// SIMATIC STEP 7 (V5.x) project BAS_20HSL
// CPU: CPU 414-5 H PN/DP(1)
// CPU: CPU 414-5 H PN/DP
// CPU: CPU 414-5 H PN/DP
// CPU: CPU 412-5 H PN/DP
// CPU: CPU 414-5 H PN/DP(1)
// station: Hardware
// station: B_PLC(MAIN)
// station: P_ADR_BUS
// station: Hardware
// station: P_ADR_BUS
// station: A_PLC
// station: IBP_PLC
// station: Hardware
// station: P_ADR_BUS
// program: S7 Program(2)
// program: S7 Program(1)
// program: S7 Program(1)
// program: S7 Program(5)
// program: S7 Program(9)

SYMBOL_TABLE
"CONTROL_DAT"	DB 1	DB 1
"MODBUS_HPARAM_PN_2"	DB 2	DB 2
"License DB"	DB 3	DB 3
"CPULINDB"	DB 30	DB 30
"SYS_Date_Time_D"	DB 34	DB 34	// 系统日期和时间设置和读取数据区
"FB200_DB"	DB 200	FB 200
"FB201_DB"	DB 201	FB 201
"MAIN-READ-SLAVE"	DB 202	DB 202
"MAIN-WRITE-SLAVE"	DB 203	DB 203
"MAIN-READ-IBP"	DB 204	DB 204
"MAIN-WRITE-IBP"	DB 205	DB 205
"DETAIL_DIAG_DB_RACK0"	DB 458	FB 315	// DB FOR SFB13
"DETAIL_DIAG_DB_RACK1"	DB 459	FB 315	// DB FOR SFB12
"DP_ERROR_RACK0"	DB 460	DB 460
"DP_ERROR_RESET_DB"	DB 461	DB 461
"DP_ERROR_FB1501"	DB 462	FB 1501
"DB_FOR_FB300"	DB 463	FB 300
"DP_VAT"	DB 464	DB 464
"DP_ERROR_RACK1"	DB 465	DB 465
"DP_ERROR1_RESET"	DB 466	DB 466
"DP_ERROR1_FB1501"	DB 467	FB 1501
"FB523_DB"	DB 523	FB 523
"LED"	DB 525	DB 525
"IDB_MODBUS"	DB 915	FB 915
"JOBLIST_DB"	DB 919	FB 919
"JOB_RESET_DB"	DB 921	FB 921
"AP_BMPSB"	DB 2005	DB 2005
"EPS21"	DB 2015	DB 2015
"E411_08_C"	DB 2025	DB 2025
"AT_AYSB4_WRITE"	DB 2033	DB 2033
"AT_AYSB4_READ"	DB 2035	DB 2035
"AT_aysb1_2_WRITE"	DB 2043	DB 2043
"AT_AYSB1_2_READ"	DB 2045	DB 2045
"AP_PSB_C1_C2"	DB 2055	DB 2055
"AT_FSB_3_4_PSD2"	DB 2065	DB 2065
"AP_PSB_C"	DB 2075	DB 2075
"EPS11"	DB 2095	DB 2095
"E411_01_02_N"	DB 2105	DB 2105
"AP_FSB_WRITE"	DB 2113	DB 2113
"AP_FSB_READ"	DB 2115	DB 2115
"AT_QJSB_WRITE"	DB 2123	DB 2123
"AT_QJSB_READ"	DB 2125	DB 2125
"HF3_IMCC_Read_DB2291"	DB 2291	DB 2291	// IMCC系统读取数据
"HF3_IMCC_Write_DB2292"	DB 2292	DB 2292	// IMCC系统写数据
"HF3_EPS_HMI"	DB 2501	FB 2501	// EPS_ToHMI
"IMCC_LOCK"	DB 2555	DB 2555
"MAIN_ToHMI"	DB 6002	DB 6002	// 发送数据至HMI
"ISCS_CONTROL"	DB 6003	DB 6003
"SLAVE_TO_HMI"	DB 6004	DB 6004
"HF3_DP_Statu_ToHMI"	DB 6009	DB 6009
"HF3_PLC_Statu_ToHMI"	DB 6010	DB 6010
"给上位_状态"	DB 6030	DB 6030
"HF4_Sum_SCtrl"	DB 6040	DB 6040
"HF4_Mode_DB"	DB 7004	DB 7004	// B端模式控制命令
"Maste_To_Slave_Mod_DB"	DB 7005	DB 7005
"MODE_REFUSE"	DB 7006	DB 7006
"P_RCV"	FB 12	FB 12	// Receive Data from CP340
"P_SEND"	FB 13	FB 13	// Send Data to CP340
"pid"	FB 41	FB 41
"TSEND"	FB 63	FB 63	// Send Data
"TRCV"	FB 64	FB 64	// Receive Data
"TCON"	FB 65	FB 65	// Connect
"TDISCON"	FB 66	FB 66	// Disconnect
"P_RESET"	FB 177	FB 177	// Reset Job for CP340
"S7400H-COM-MAIN-SLAVE"	FB 200	FB 200
"S7400H-COM-MAIN-IBP"	FB 201	FB 201
"S7400H-COM-SLAVE-MAIN"	FB 202	FB 202
"READ_ERROR"	FB 300	FB 300
"DETAIL_DP_DIAG"	FB 315	FB 315
"H_STATUS"	FB 523	FB 523	// Status H-System
"TCP_COMM"	FB 913	FB 913	// TCP Kommunikation
"MOD_CLI"	FB 914	FB 914
"MB_PNHCL"	FB 915	FB 915
"Job_List"	FB 919	FB 919
"JOB_RESET"	FB 921	FB 921
"MODMAS_STEP7_CP340_L"	FB 1071	FB 1071
"com_check"	FB 1501	FB 1501
"HF3_PID_FB2005"	FB 2005	FB 2005	// PID处理功能块
"HF3_RunFaultSum"	FB 2006	FB 2006	// 运行时间故障次数统计
"HF3_EPS_FB2501"	FB 2501	FB 2501	// EPS主程序段
"HF3_EPS_FB2502"	FB 2502	FB 2502	// EPS功能块
"HF3_IMCC_CommOK_FB2512"	FB 2512	FB 2512	// IMCC心跳
"HF3_IMCC_CommOK_FB2513"	FB 2513	FB 2513
"HF3_LSQK_FB2521"	FB 2521	FB 2521	// 冷水群控程序段
"HF3_LSQK_FB2522"	FB 2522	FB 2522	// LSQK功能块
"HF3_JET_FB2531"	FB 2531	FB 2531	// 射流风机主程序端
"HF3_JET_FB2532"	FB 2532	FB 2532	// 射流风机功能块
"HF3_VRV_FB2541"	FB 2541	FB 2541	// 多联体空调主程序段
"HF3_VRV_FB2542"	FB 2542	FB 2542	// 多联体空调程序端
"HF3_SB_FB2551"	FB 2551	FB 2551	// 带控制水泵程序段
"HF3_SB_FB2552"	FB 2552	FB 2552	// 带控制水泵功能块
"HF3_3#SB_FB2561"	FB 2561	FB 2561	// 洞口水泵主程序段
"HF3_3#SB_FB2562"	FB 2562	FB 2562	// 洞口水泵功能块
"HF3_WSB_FB2581"	FB 2581	FB 2581	// 污水密闭提升
"HF3_WSB_FB2582"	FB 2582	FB 2582
"HF3_PSB_FB2591"	FB 2591	FB 2591	// 局部排水泵主程序
"HF3_PSB_FB2592"	FB 2592	FB 2592	// 排水泵DB转换
"HF3_UPS_FB2611"	FB 2611	FB 2611
"HF3_UPS_FB2612"	FB 2612	FB 2612
"HF3_DT_FB2621"	FB 2621	FB 2621	// 电梯
"HF3_DT_FB2622"	FB 2622	FB 2622	// 电梯
"HF3_FT_FB2631"	FB 2631	FB 2631	// 扶梯
"HF4_FT_FB2362"	FB 2632	FB 2632
"HF3_IMCC_TVF_FB2651"	FB 2651	FB 2651	// 隧道风机主程序段
"HF4_IMCC_TVF_FB2652"	FB 2652	FB 2652	// 隧道风机功能块
"HF3_IMCC_TEF_FB2661"	FB 2661	FB 2661	// 排热风机主程序
"HF3_IMCC_TEF_FB2662"	FB 2662	FB 2662	// 排热风机功能块
"HF3_IMCC_KT_FB2671"	FB 2671	FB 2671	// 大空调主程序
"HF3_IMCC_KT_FB2672"	FB 2672	FB 2672	// 空调机组功能块
"HF3_IMCC_HPF_FB2681"	FB 2681	FB 2681	// IMCC_HPF_主程序
"HF4_IMCC_HPF_FB2682"	FB 2682	FB 2682	// IMCC_HPF功能块
"HF3_IMCC_FJ_FB2691"	FB 2691	FB 2691	// 智能低压小风机
"HF3_IMCC_FJ_FB2692"	FB 2692	FB 2692	// 智能低压小风机功能块
"HF3_IMCC_DZ_FB2701"	FB 2701	FB 2701	// IMCC组合阀主程序
"HF3_IMCC_DZ_B2702"	FB 2702	FB 2702	// 电动组合风阀功能块
"HF3_IMCC_DT_FB2711"	FB 2711	FB 2711	// IMCC风量调节阀程序
"HF3_IMCC_DT_FB2712"	FB 2712	FB 2712	// IMCC风量调节阀块
"HF3_IMCC_D_FB2721"	FB 2721	FB 2721	// IMCC电动风阀主程序
"HF3_IMCC_D_FB2722"	FB 2722	FB 2722	// IMCC电动风阀功能块
"HF3_JH_YC_FB2731"	FB 2731	FB 2731	// 电子净化压差主程序
"HF3_DPH_FB2751"	FB 2751	FB 2751	// 二通阀主程序
"HF3_DPH_FB2752"	FB 2752	FB 2752	// 二通阀主程序
"HF3_FJ_FB2761"	FB 2761	FB 2761	// 高架站风机主程序段
"HF3_FJ_FB2762"	FB 2762	FB 2762	// 高架站风机
"HF3_FJPG_FB2771"	FB 2771	FB 2771	// 风机盘管主程序段
"HF3_FJPG_FB2772"	FB 2772	FB 2772	// 风机盘管功能块
"HF3_XFDF_FB2781"	FB 2781	FB 2781	// 手电一体蝶阀程序段
"HF2_XVDF_FB2782"	FB 2782	FB 2782	// 手电一体蝶阀功能块
"HF3_EPS_WLE_FB2791"	FB 2791	FB 2791	// 区间疏散指示
"HF3_EPS_WLE_FB2792"	FB 2792	FB 2792	// 区间疏散指示功能块
"HF3_D_FB2801"	FB 2801	FB 2801	// 高架站风阀主程序
"HF3_D_FB2802"	FB 2802	FB 2802	// 高架站风阀功能块
"HF3_FHF_RFM_FB2811"	FB 2811	FB 2811	// 防火阀人防门
"HF3_Senor_FB2821"	FB 2821	FB 2821	// 传感器程序段
"HF3_Sensor_FB2822"	FB 2822	FB 2822	// 传感器功能块
"AB_IBP_Comm"	FB 2831	FB 2831
"从端与主端通讯"	FB 2832	FB 2832
"HF3_MODE_PRO"	FB 3000	FB 3000
"HF3_Mode_Explode_FB3005"	FB 3005	FB 3005	// 模式表分解
"HF3_Mode_Explode_FB3019"	FB 3020	FB 3020
"IMCC_Pro"	FC 1	FC 1	// 智能低压通信数据段
"HF3_B_T_W_FC51"	FC 51	FC 51	// BOOLתWORD
"HF3_W_T_B_FC54"	FC 54	FC 54	// WORDתBOOL
"SCALE"	FC 105	FC 105	// Scaling Values
"UNSCALE"	FC 106	FC 106	// Unscaling Values
"MK_ERROR_SAVE_RACK0"	FC 201	FC 201
"RIO_Information"	FC 202	FC 202
"MK_ERROR_SAVE_RACK1"	FC 203	FC 203
"DP_ERROR_TO_DB701"	FC 204	FC 204
"GET_DBN"	FC 501	FC 501	// Get DB Nummer
"BAS_CLOCK"	FC 505	FC 505
"CPU_Information"	FC 523	FC 523
"ABS_I"	FC 1234	FC 1234
"real_to_int"	FC 2000	FC 2000
"HF3_IMCC_FC2511"	FC 2511	FC 2511
"HF3_Mode_Refuse_FC3011"	FC 3011	FC 3011
"FUZHI"	FC 4000	FC 4000
"HF3_CP340_FC4301"	FC 4301	FC 4301	// CP340_配置程序段
"SDPH_A1_LR"	I 0.0	BOOL	// 远程/就地状态
"SDPH_K4_A1_LR"	I 0.1	BOOL	// 远程/就地状态
"YC_A_Alarm"	I 0.2	BOOL	// 压差开关报警
"JH_A_Run"	I 0.3	BOOL	// 运行信号
"JH_A_Stp"	I 0.4	BOOL	// 停止信号
"JH_A_Wash"	I 0.5	BOOL	// 清洗信号
"JH_A_Flt"	I 0.6	BOOL	// 综合故障报警信号
"JH_A_Auto"	I 0.7	BOOL	// 自动/手动信号
"EPS11_QJSS_UEF_Opd"	I 2.0	BOOL	// 上行头前向反馈
"EPS11_QJSS_UEB_Opd"	I 2.1	BOOL	// 上行头后向反馈
"EPS11_QJSS_DHF_Opd"	I 2.2	BOOL	// 下行尾前向反馈
"EPS11_QJSS_DHB_opd"	I 2.3	BOOL	// 下行尾后向反馈
"Always0"	M 0.0	BOOL	// 保持0
"Always1"	M 0.1	BOOL	// 保持1
"IMCC_Comok"	M 50.0	BOOL
"ABC"	M 50.1	BOOL
"JOB_PLUS"	M 100.0	BOOL
"HF3_Main_OB1"	OB 1	OB 1	// 程序主循环
"CYC_INT5"	OB 35	OB 35	// Cyclic Interrupt 5
"RED_I/O_FLT1"	OB 70	OB 70	// Redundancy I/O Fault 1
"RED_FLT"	OB 72	OB 72	// Redundancy Fault
"PS_FLT"	OB 81	OB 81	// Power Supply Fault
"I/O_FLT1"	OB 82	OB 82	// I/O ZOint Fault 1
"I/O_FLT2"	OB 83	OB 83	// I/O Point Fault 2
"CPU_FLT"	OB 84	OB 84	// CPU Fault
"OBNL_FLT"	OB 85	OB 85	// OB Not Loaded Fault
"RACK_FLT"	OB 86	OB 86	// Loss of Rack Fault
"COMM_FLT"	OB 87	OB 87	// Communication Fault
"COMPLETE RESTART"	OB 100	OB 100	// Complete Restart
"PROG_ERR"	OB 121	OB 121	// Programming Error
"MOD_ERR"	OB 122	OB 122	// Module Access Error
"H_A4_aiHumi"	PIW 512	INT	// 湿度反馈
"H_A4_aiTemp"	PIW 514	INT	// 温度反馈
"H_A5_aiHumi"	PIW 516	INT	// 湿度反馈
"H_A5_aiTemp"	PIW 518	INT	// 温度反馈
"C_A3_aiCO2"	PIW 524	INT	// 二氧化碳浓度反馈
"K4_T_A1_aiHumi"	PIW 528	INT	// 湿度反馈
"K4_T_A1_aiTemp"	PIW 530	INT	// 温度反馈
"H_A2_aiHumi"	PIW 544	INT	// 湿度反馈
"H_A2_aiTemp"	PIW 546	INT	// 温度反馈
"H_A3_aiHumi"	PIW 548	INT	// 湿度反馈
"H_A3_aiTemp"	PIW 550	INT	// 温度反馈
"K4_H_A1_aiHumi"	PIW 552	INT	// 湿度反馈
"K4_H_A1_aiTemp"	PIW 554	INT	// 温度反馈
"H_A1_aiHumi"	PIW 556	INT	// 湿度反馈
"H_A1_aiTemp"	PIW 558	INT	// 温度反馈
"SDPH_K4_A1_aiPFB"	PIW 568	INT	// 开度反馈
"SDPH_A_aiPFB"	PIW 570	INT	// 开度反馈
"H_A6_aiHumi"	PIW 576	INT	// 湿度反馈
"H_A6_aiTemp"	PIW 578	INT	// 温度反馈
"H_A7_aiHumi"	PIW 580	INT	// 湿度反馈
"H_A7_aiTemp"	PIW 582	INT	// 温度反馈
"C_A2_aiCO2"	PIW 588	INT	// 二氧化碳浓度反馈
"C_A4_aiCO2"	PIW 590	INT	// 二氧化碳浓度反馈
"T_A2_aiHumi"	PIW 592	INT	// 湿度反馈
"T_A2_aiTemp"	PIW 594	INT	// 温度反馈
"SDPH_A1_aqPset"	PQW 512	INT	// 开度控制
"SDPH_K4_A1_aqPset"	PQW 514	INT	// 开度控制
"EPS11_QJSS_UEF_opn"	Q 0.0	BOOL	// 上行头前向控制
"EPS11_QJSS_UEB_opn"	Q 0.1	BOOL	// 上行头后向控制
"EPS11_QJSS_DHF_opn"	Q 0.2	BOOL	// 下行尾前向控制
"EPS11_QJSS_DHB_opn"	Q 0.3	BOOL	// 下行尾后向控制
"TON"	SFB 4	SFB 4	// Generate an On Delay
"BSEND"	SFB 12	SFB 12	// Sending Segmented Data
"BRCV"	SFB 13	SFB 13	// Receiving Segmented Data
"ALARM_8P"	SFB 35	SFB 35	// Generate Block-Related Messages with Values for 8 Signals
"RDREC"	SFB 52	SFB 52	// Read a Process Data Record
"WRREC"	SFB 53	SFB 53	// Write a Process Data Record
"READ_CLK"	SFC 1	SFC 1	// Read System Clock
"GADR_LGC"	SFC 5	SFC 5	// Query Logical Address of a Channel
"RD_SINFO"	SFC 6	SFC 6	// Read OB Start Information
"DPNRM_DG"	SFC 13	SFC 13	// Read Diagnostic Data of a DP Slave
"BLKMOV"	SFC 20	SFC 20	// Copy Variables
"TEST_DB"	SFC 24	SFC 24	// Test Data Block
"DIS_AIRT"	SFC 41	SFC 41	// Delay the Higher Priority Interrupts and Asynchronous Errors
"EN_AIRT"	SFC 42	SFC 42	// Enable Higher Priority Interrupts and Asynchronous Errors
"LGC_GADR"	SFC 49	SFC 49	// Query the Module Slot Belonging to a Logical Address
"RDSYSST"	SFC 51	SFC 51	// Read a System Status List or Partial List
"WR_REC"	SFC 58	SFC 58	// Write Data Record
"RD_REC"	SFC 59	SFC 59	// Read a Data Record
"T800"	T 800	TIMER
"UDT_ANY_Pointer"	UDT 10	UDT 10
"VAT_1"	VAT 1	
"Client_Job"	VAT 6	
END_SYMBOL_TABLE

TYPE "UDT_ANY_Pointer"	// UDT 10
VERSION : 0.0
  STRUCT
   Syntax_ID : BYTE ;
   DataTyp : BYTE ;
   Count : WORD ;
   DB_Number : WORD ;
   Byte_Pointer : DWORD ;
  END_STRUCT ;	
END_TYPE

// FB 12: know-how protected block, not included

// FB 13: know-how protected block, not included

// FB 41: know-how protected block, not included

// FB 63: know-how protected block, not included

// FB 64: know-how protected block, not included

// FB 65: know-how protected block, not included

// FB 66: know-how protected block, not included

// FB 177: know-how protected block, not included

FUNCTION_BLOCK "S7400H-COM-MAIN-IBP"	// FB 201
VERSION : 0.1
VAR_OUTPUT
  STATUS_1 : BOOL ;
  STATUS_2 : BOOL ;
END_VAR
VAR
  BSEND_1 : SFB 12;
  BSEND_2 : SFB 12;
  BREV_1 : SFB 13;
  BREV_2 : SFB 13;
  LENTH : WORD ;
  TON_1 : SFB 4;
  TON_2 : SFB 4;
END_VAR
BEGIN
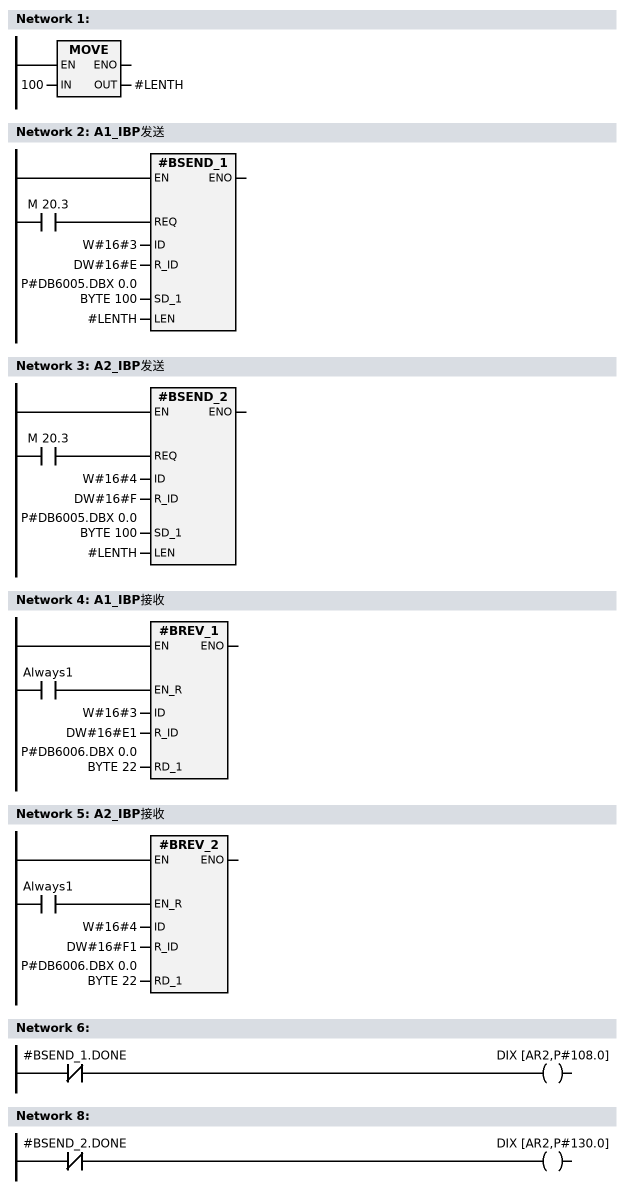
NETWORK
TITLE =
      L     100;
      T     #LENTH;
      NOP   0;
NETWORK
TITLE = A1_IBP发送
      A     M 20.3;
      =     L 0.0;
      BLD   103;
      CALL  #BSEND_1 (
           REQ                      := L 0.0,
           ID                       := W#16#3,
           R_ID                     := DW#16#E,
           SD_1                     := P#DB6005.DBX 0.0 BYTE 100,
           LEN                      := #LENTH);
      NOP   0;
NETWORK
TITLE = A2_IBP发送
      A     M 20.3;
      =     L 0.0;
      BLD   103;
      CALL  #BSEND_2 (
           REQ                      := L 0.0,
           ID                       := W#16#4,
           R_ID                     := DW#16#F,
           SD_1                     := P#DB6005.DBX 0.0 BYTE 100,
           LEN                      := #LENTH);
      NOP   0;
NETWORK
TITLE = A1_IBP接收
      A     "Always1";
      =     L 0.0;
      BLD   103;
      CALL  #BREV_1 (
           EN_R                     := L 0.0,
           ID                       := W#16#3,
           R_ID                     := DW#16#E1,
           RD_1                     := P#DB6006.DBX 0.0 BYTE 22);
      NOP   0;
NETWORK
TITLE = A2_IBP接收
      A     "Always1";
      =     L 0.0;
      BLD   103;
      CALL  #BREV_2 (
           EN_R                     := L 0.0,
           ID                       := W#16#4,
           R_ID                     := DW#16#F1,
           RD_1                     := P#DB6006.DBX 0.0 BYTE 22);
      NOP   0;
NETWORK
TITLE =
      AN    #BSEND_1.DONE;
      =     DIX [AR2,P#108.0];
NETWORK
TITLE =
      BLD   16;
      =     L 7.0;
      L     DINO;
      T     LW 5;
      CDB;
      OPN   DI [LW 5];
      TAR2  LD 1;
      L     L#5000;
      T     DID [AR2,P#110.0];
      +AR2  P#108.0;
      UC    "TON";
      LAR2  LD 1;
      A     DIX [AR2,P#114.0];
      =     DBX [AR2,P#0.0];
      CDB;
      BLD   17;
      NOP   0;
NETWORK
TITLE =
      AN    #BSEND_2.DONE;
      =     DIX [AR2,P#130.0];
NETWORK
TITLE =
      BLD   16;
      =     L 7.0;
      L     DINO;
      T     LW 5;
      CDB;
      OPN   DI [LW 5];
      TAR2  LD 1;
      L     L#5000;
      T     DID [AR2,P#132.0];
      +AR2  P#130.0;
      UC    "TON";
      LAR2  LD 1;
      A     DIX [AR2,P#136.0];
      =     DBX [AR2,P#0.1];
      CDB;
      BLD   17;
      NOP   0;
END_FUNCTION_BLOCK

FUNCTION_BLOCK "S7400H-COM-SLAVE-MAIN"	// FB 202
VERSION : 0.1
VAR_OUTPUT
  STATUS_1 : BOOL ;
  STATUS_2 : BOOL ;
END_VAR
VAR
  BSEND_1 : SFB 12;
  BSEND_2 : SFB 12;
  BSEND_3 : SFB 12;
  BSEND_4 : SFB 12;
  BREV_1 : SFB 13;
  BREV_2 : SFB 13;
  BREV_3 : SFB 13;
  BREV_4 : SFB 13;
  LENTH1 : WORD ;
  LENTH2 : WORD ;
  TON_1 : SFB 4;
  TON_2 : SFB 4;
  stat_SEND1 : SFB 12;
  stat_SEND2 : SFB 12;
  stat_SEND3 : SFB 12;
  stat_SEND4 : SFB 12;
  LENTH3 : WORD ;
  LENTH4 : WORD ;
END_VAR
BEGIN
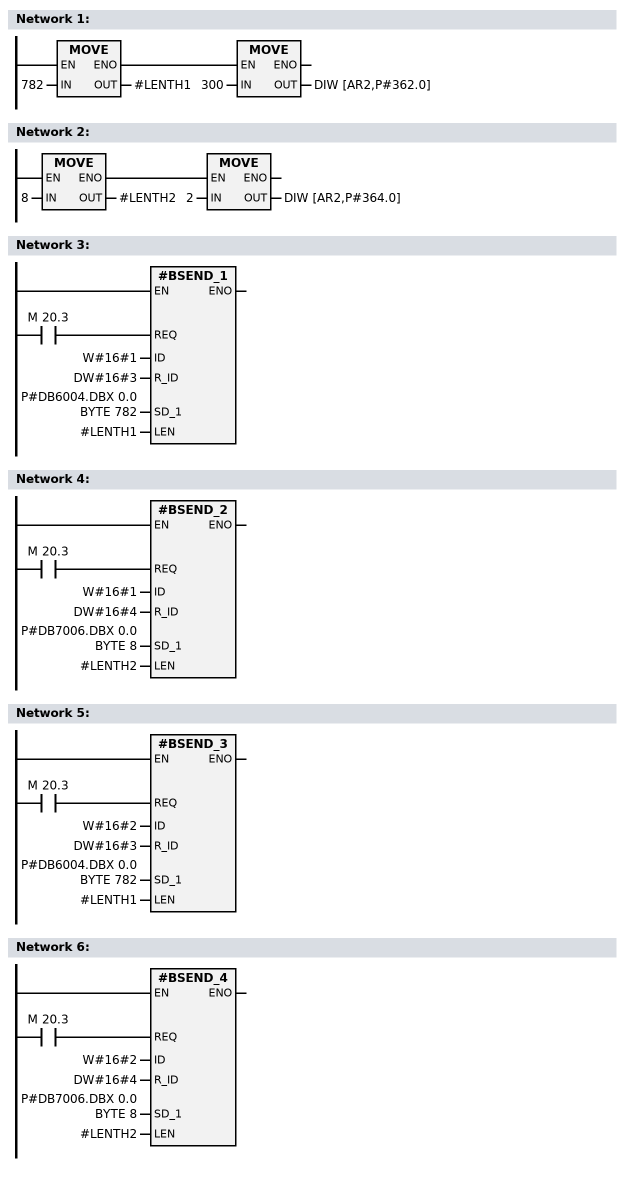
NETWORK
TITLE =
      A(;
      L     782;
      T     #LENTH1;
      SET;
      SAVE;
      CLR;
      A     BR;
      );
      JNB   _001;
      L     300;
      T     DIW [AR2,P#362.0];
_001: NOP   0;
NETWORK
TITLE =
      A(;
      L     8;
      T     #LENTH2;
      SET;
      SAVE;
      CLR;
      A     BR;
      );
      JNB   _002;
      L     2;
      T     DIW [AR2,P#364.0];
_002: NOP   0;
NETWORK
TITLE =
      A     M 20.3;
      =     L 0.0;
      BLD   103;
      CALL  #BSEND_1 (
           REQ                      := L 0.0,
           ID                       := W#16#1,
           R_ID                     := DW#16#3,
           SD_1                     := P#DB6004.DBX 0.0 BYTE 782,
           LEN                      := #LENTH1);
      NOP   0;
NETWORK
TITLE =
      A     M 20.3;
      =     L 0.0;
      BLD   103;
      CALL  #BSEND_2 (
           REQ                      := L 0.0,
           ID                       := W#16#1,
           R_ID                     := DW#16#4,
           SD_1                     := P#DB7006.DBX 0.0 BYTE 8,
           LEN                      := #LENTH2);
      NOP   0;
NETWORK
TITLE =
      A     M 20.3;
      =     L 0.0;
      BLD   103;
      CALL  #BSEND_3 (
           REQ                      := L 0.0,
           ID                       := W#16#2,
           R_ID                     := DW#16#3,
           SD_1                     := P#DB6004.DBX 0.0 BYTE 782,
           LEN                      := #LENTH1);
      NOP   0;
NETWORK
TITLE =
      A     M 20.3;
      =     L 0.0;
      BLD   103;
      CALL  #BSEND_4 (
           REQ                      := L 0.0,
           ID                       := W#16#2,
           R_ID                     := DW#16#4,
           SD_1                     := P#DB7006.DBX 0.0 BYTE 8,
           LEN                      := #LENTH2);
      NOP   0;
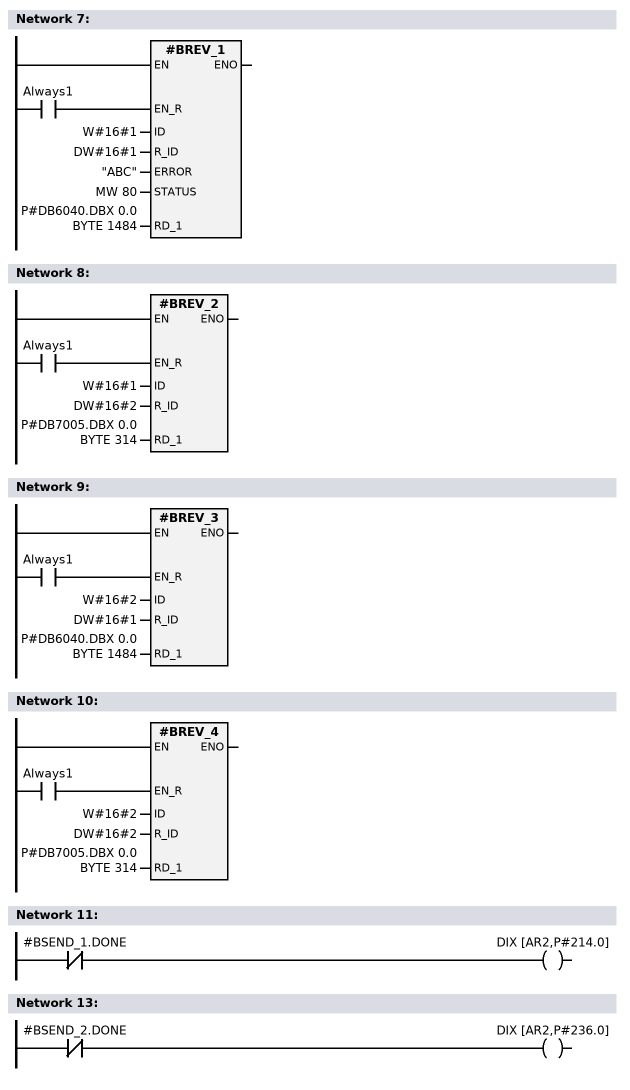
NETWORK
TITLE =
      A     "Always1";
      =     L 0.0;
      BLD   103;
      CALL  #BREV_1 (
           EN_R                     := L 0.0,
           ID                       := W#16#1,
           R_ID                     := DW#16#1,
           ERROR                    := "ABC",
           STATUS                   := MW 80,
           RD_1                     := P#DB6040.DBX 0.0 BYTE 1484);
      NOP   0;
NETWORK
TITLE =
      A     "Always1";
      =     L 0.0;
      BLD   103;
      CALL  #BREV_2 (
           EN_R                     := L 0.0,
           ID                       := W#16#1,
           R_ID                     := DW#16#2,
           RD_1                     := P#DB7005.DBX 0.0 BYTE 314);
      NOP   0;
NETWORK
TITLE =
      A     "Always1";
      =     L 0.0;
      BLD   103;
      CALL  #BREV_3 (
           EN_R                     := L 0.0,
           ID                       := W#16#2,
           R_ID                     := DW#16#1,
           RD_1                     := P#DB6040.DBX 0.0 BYTE 1484);
      NOP   0;
NETWORK
TITLE =
      A     "Always1";
      =     L 0.0;
      BLD   103;
      CALL  #BREV_4 (
           EN_R                     := L 0.0,
           ID                       := W#16#2,
           R_ID                     := DW#16#2,
           RD_1                     := P#DB7005.DBX 0.0 BYTE 314);
      NOP   0;
NETWORK
TITLE =
      AN    #BSEND_1.DONE;
      =     DIX [AR2,P#214.0];
NETWORK
TITLE =
      BLD   16;
      =     L 7.0;
      L     DINO;
      T     LW 5;
      CDB;
      OPN   DI [LW 5];
      TAR2  LD 1;
      L     L#5000;
      T     DID [AR2,P#216.0];
      +AR2  P#214.0;
      UC    "TON";
      LAR2  LD 1;
      A     DIX [AR2,P#220.0];
      =     DBX [AR2,P#0.0];
      CDB;
      BLD   17;
      NOP   0;
NETWORK
TITLE =
      AN    #BSEND_2.DONE;
      =     DIX [AR2,P#236.0];
NETWORK
TITLE =
      BLD   16;
      =     L 7.0;
      L     DINO;
      T     LW 5;
      CDB;
      OPN   DI [LW 5];
      TAR2  LD 1;
      L     L#5000;
      T     DID [AR2,P#238.0];
      +AR2  P#236.0;
      UC    "TON";
      LAR2  LD 1;
      A     DIX [AR2,P#242.0];
      =     DBX [AR2,P#0.1];
      CDB;
      BLD   17;
      NOP   0;
NETWORK
TITLE =
      A     M 20.3;
      =     L 0.0;
      BLD   103;
      BLD   16;
      =     L 7.0;
      L     DINO;
      T     LW 5;
      CDB;
      OPN   DI [LW 5];
      TAR2  LD 1;
      A     L 0.0;
      =     DIX [AR2,P#258.0];
      L     1;
      T     DIW [AR2,P#260.0];
      L     L#10;
      T     DID [AR2,P#262.0];
      L     W#16#1002;
      T     DIW [AR2,P#270.0];
      L     300;
      T     DIW [AR2,P#272.0];
      L     6009;
      T     DIW [AR2,P#274.0];
      L     P#DBX 0.0;
      T     DID [AR2,P#276.0];
      L     DBW [AR2,P#362.0];
      T     DIW [AR2,P#280.0];
      +AR2  P#258.0;
      UC    "BSEND";
      LAR2  LD 1;
      L     DIW [AR2,P#280.0];
      T     DBW [AR2,P#362.0];
      CDB;
      BLD   17;
      NOP   0;
NETWORK
TITLE =
      A     M 20.3;
      =     L 0.0;
      BLD   103;
      BLD   16;
      =     L 7.0;
      L     DINO;
      T     LW 5;
      CDB;
      OPN   DI [LW 5];
      TAR2  LD 1;
      A     L 0.0;
      =     DIX [AR2,P#284.0];
      L     1;
      T     DIW [AR2,P#286.0];
      L     L#11;
      T     DID [AR2,P#288.0];
      L     W#16#1002;
      T     DIW [AR2,P#296.0];
      L     2;
      T     DIW [AR2,P#298.0];
      L     6010;
      T     DIW [AR2,P#300.0];
      L     P#DBX 0.0;
      T     DID [AR2,P#302.0];
      L     DBW [AR2,P#364.0];
      T     DIW [AR2,P#306.0];
      +AR2  P#284.0;
      UC    "BSEND";
      LAR2  LD 1;
      L     DIW [AR2,P#306.0];
      T     DBW [AR2,P#364.0];
      CDB;
      BLD   17;
      NOP   0;
NETWORK
TITLE =
      A     M 20.3;
      =     L 0.0;
      BLD   103;
      BLD   16;
      =     L 7.0;
      L     DINO;
      T     LW 5;
      CDB;
      OPN   DI [LW 5];
      TAR2  LD 1;
      A     L 0.0;
      =     DIX [AR2,P#310.0];
      L     2;
      T     DIW [AR2,P#312.0];
      L     L#10;
      T     DID [AR2,P#314.0];
      L     W#16#1002;
      T     DIW [AR2,P#322.0];
      L     300;
      T     DIW [AR2,P#324.0];
      L     6009;
      T     DIW [AR2,P#326.0];
      L     P#DBX 0.0;
      T     DID [AR2,P#328.0];
      L     DBW [AR2,P#362.0];
      T     DIW [AR2,P#332.0];
      +AR2  P#310.0;
      UC    "BSEND";
      LAR2  LD 1;
      L     DIW [AR2,P#332.0];
      T     DBW [AR2,P#362.0];
      CDB;
      BLD   17;
      NOP   0;
NETWORK
TITLE =
      A     M 20.3;
      =     L 0.0;
      BLD   103;
      BLD   16;
      =     L 7.0;
      L     DINO;
      T     LW 5;
      CDB;
      OPN   DI [LW 5];
      TAR2  LD 1;
      A     L 0.0;
      =     DIX [AR2,P#336.0];
      L     2;
      T     DIW [AR2,P#338.0];
      L     L#11;
      T     DID [AR2,P#340.0];
      L     W#16#1002;
      T     DIW [AR2,P#348.0];
      L     2;
      T     DIW [AR2,P#350.0];
      L     6010;
      T     DIW [AR2,P#352.0];
      L     P#DBX 0.0;
      T     DID [AR2,P#354.0];
      L     DBW [AR2,P#364.0];
      T     DIW [AR2,P#358.0];
      +AR2  P#336.0;
      UC    "BSEND";
      LAR2  LD 1;
      L     DIW [AR2,P#358.0];
      T     DBW [AR2,P#364.0];
      CDB;
      BLD   17;
      NOP   0;
END_FUNCTION_BLOCK

FUNCTION_BLOCK "READ_ERROR"	// FB 300
VERSION : 0.1
VAR_TEMP
  MID1 : BOOL ;
  MID11 : INT ;
  MID2 : BOOL ;
  MID22 : INT ;
END_VAR
BEGIN
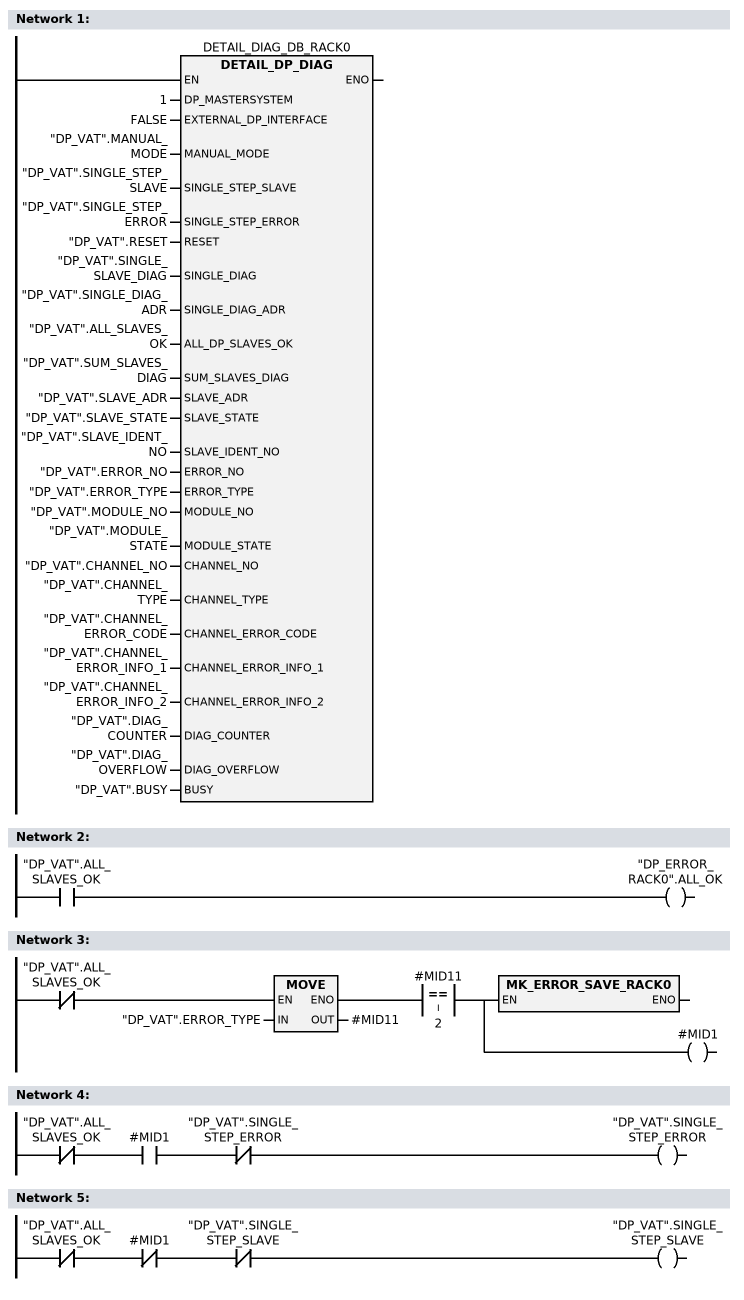
NETWORK
TITLE =
//DP_MASTERSYSTEM=1
      CALL  "DETAIL_DP_DIAG" , "DETAIL_DIAG_DB_RACK0" (
           DP_MASTERSYSTEM          := 1,
           EXTERNAL_DP_INTERFACE    := FALSE,
           MANUAL_MODE              := "DP_VAT".MANUAL_MODE,
           SINGLE_STEP_SLAVE        := "DP_VAT".SINGLE_STEP_SLAVE,
           SINGLE_STEP_ERROR        := "DP_VAT".SINGLE_STEP_ERROR,
           RESET                    := "DP_VAT".RESET,
           SINGLE_DIAG              := "DP_VAT".SINGLE_SLAVE_DIAG,
           SINGLE_DIAG_ADR          := "DP_VAT".SINGLE_DIAG_ADR,
           ALL_DP_SLAVES_OK         := "DP_VAT".ALL_SLAVES_OK,
           SUM_SLAVES_DIAG          := "DP_VAT".SUM_SLAVES_DIAG,
           SLAVE_ADR                := "DP_VAT".SLAVE_ADR,
           SLAVE_STATE              := "DP_VAT".SLAVE_STATE,
           SLAVE_IDENT_NO           := "DP_VAT".SLAVE_IDENT_NO,
           ERROR_NO                 := "DP_VAT".ERROR_NO,
           ERROR_TYPE               := "DP_VAT".ERROR_TYPE,
           MODULE_NO                := "DP_VAT".MODULE_NO,
           MODULE_STATE             := "DP_VAT".MODULE_STATE,
           CHANNEL_NO               := "DP_VAT".CHANNEL_NO,
           CHANNEL_TYPE             := "DP_VAT".CHANNEL_TYPE,
           CHANNEL_ERROR_CODE       := "DP_VAT".CHANNEL_ERROR_CODE,
           CHANNEL_ERROR_INFO_1     := "DP_VAT".CHANNEL_ERROR_INFO_1,
           CHANNEL_ERROR_INFO_2     := "DP_VAT".CHANNEL_ERROR_INFO_2,
           DIAG_COUNTER             := "DP_VAT".DIAG_COUNTER,
           DIAG_OVERFLOW            := "DP_VAT".DIAG_OVERFLOW,
           BUSY                     := "DP_VAT".BUSY);
      NOP   0;
NETWORK
TITLE =
      A     "DP_VAT".ALL_SLAVES_OK;
      =     "DP_ERROR_RACK0".ALL_OK;
NETWORK
TITLE =
      A(;
      AN    "DP_VAT".ALL_SLAVES_OK;
      JNB   _001;
      L     "DP_VAT".ERROR_TYPE;
      T     #MID11;
      SET;
      SAVE;
      CLR;
_001: A     BR;
      );
      A(;
      L     #MID11;
      L     2;
      ==I;
      );
      =     L 8.0;
      A     L 8.0;
      JNB   _002;
      CALL  "MK_ERROR_SAVE_RACK0";
_002: NOP   0;
      A     L 8.0;
      BLD   102;
      =     #MID1;
NETWORK
TITLE =
      AN    "DP_VAT".ALL_SLAVES_OK;
      A     #MID1;
      AN    "DP_VAT".SINGLE_STEP_ERROR;
      =     "DP_VAT".SINGLE_STEP_ERROR;
NETWORK
TITLE =
      AN    "DP_VAT".ALL_SLAVES_OK;
      AN    #MID1;
      AN    "DP_VAT".SINGLE_STEP_SLAVE;
      =     "DP_VAT".SINGLE_STEP_SLAVE;
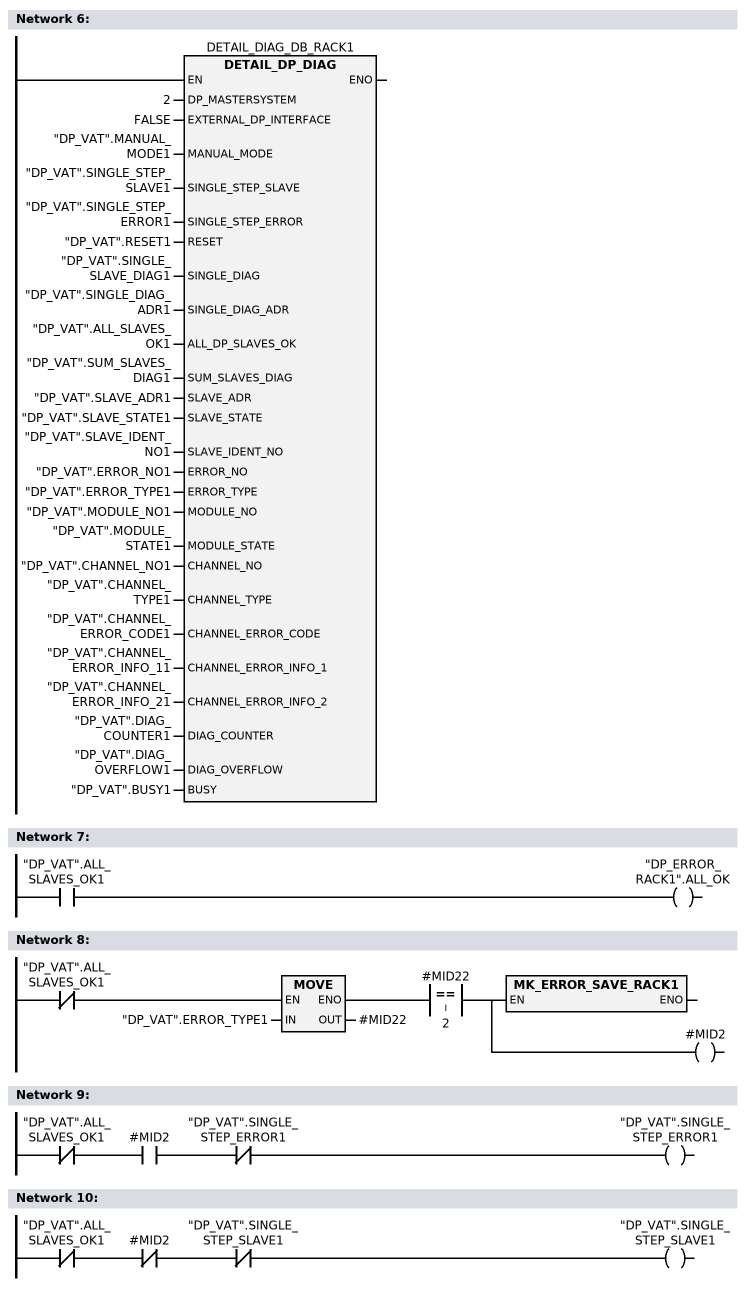
NETWORK
TITLE =
//DP_MASTERSYSTEM=2
      CALL  "DETAIL_DP_DIAG" , "DETAIL_DIAG_DB_RACK1" (
           DP_MASTERSYSTEM          := 2,
           EXTERNAL_DP_INTERFACE    := FALSE,
           MANUAL_MODE              := "DP_VAT".MANUAL_MODE1,
           SINGLE_STEP_SLAVE        := "DP_VAT".SINGLE_STEP_SLAVE1,
           SINGLE_STEP_ERROR        := "DP_VAT".SINGLE_STEP_ERROR1,
           RESET                    := "DP_VAT".RESET1,
           SINGLE_DIAG              := "DP_VAT".SINGLE_SLAVE_DIAG1,
           SINGLE_DIAG_ADR          := "DP_VAT".SINGLE_DIAG_ADR1,
           ALL_DP_SLAVES_OK         := "DP_VAT".ALL_SLAVES_OK1,
           SUM_SLAVES_DIAG          := "DP_VAT".SUM_SLAVES_DIAG1,
           SLAVE_ADR                := "DP_VAT".SLAVE_ADR1,
           SLAVE_STATE              := "DP_VAT".SLAVE_STATE1,
           SLAVE_IDENT_NO           := "DP_VAT".SLAVE_IDENT_NO1,
           ERROR_NO                 := "DP_VAT".ERROR_NO1,
           ERROR_TYPE               := "DP_VAT".ERROR_TYPE1,
           MODULE_NO                := "DP_VAT".MODULE_NO1,
           MODULE_STATE             := "DP_VAT".MODULE_STATE1,
           CHANNEL_NO               := "DP_VAT".CHANNEL_NO1,
           CHANNEL_TYPE             := "DP_VAT".CHANNEL_TYPE1,
           CHANNEL_ERROR_CODE       := "DP_VAT".CHANNEL_ERROR_CODE1,
           CHANNEL_ERROR_INFO_1     := "DP_VAT".CHANNEL_ERROR_INFO_11,
           CHANNEL_ERROR_INFO_2     := "DP_VAT".CHANNEL_ERROR_INFO_21,
           DIAG_COUNTER             := "DP_VAT".DIAG_COUNTER1,
           DIAG_OVERFLOW            := "DP_VAT".DIAG_OVERFLOW1,
           BUSY                     := "DP_VAT".BUSY1);
      NOP   0;
NETWORK
TITLE =
      A     "DP_VAT".ALL_SLAVES_OK1;
      =     "DP_ERROR_RACK1".ALL_OK;
NETWORK
TITLE =
      A(;
      AN    "DP_VAT".ALL_SLAVES_OK1;
      JNB   _003;
      L     "DP_VAT".ERROR_TYPE1;
      T     #MID22;
      SET;
      SAVE;
      CLR;
_003: A     BR;
      );
      A(;
      L     #MID22;
      L     2;
      ==I;
      );
      =     L 8.0;
      A     L 8.0;
      JNB   _004;
      CALL  "MK_ERROR_SAVE_RACK1";
_004: NOP   0;
      A     L 8.0;
      BLD   102;
      =     #MID2;
NETWORK
TITLE =
      AN    "DP_VAT".ALL_SLAVES_OK1;
      A     #MID2;
      AN    "DP_VAT".SINGLE_STEP_ERROR1;
      =     "DP_VAT".SINGLE_STEP_ERROR1;
NETWORK
TITLE =
      AN    "DP_VAT".ALL_SLAVES_OK1;
      AN    #MID2;
      AN    "DP_VAT".SINGLE_STEP_SLAVE1;
      =     "DP_VAT".SINGLE_STEP_SLAVE1;
END_FUNCTION_BLOCK

FUNCTION_BLOCK "DETAIL_DP_DIAG"	// FB 315
TITLE = DP-Diagnose / DP-Diagnosis
//Dieser Baustein wertet die Diagnose eines Profibus-DP-Systems mit S7-Master 
//aus. Der Baustein muss in den Ablaufebenen OB1, OB82 und OB86 aufgerufen 
//werden. Die Nummer des zugehoerigen Instanzdatenbausteins ist beliebig. 
//Der Aufruf des FBs in den einzelnen Ablaufebenen muss identisch sein 
//(DB-Nr, Parameterleiste). 
//Waehrend der FB-Bearbeitung werden alle Interrupts verzoegert. 
//
//This function block evaluates a Profibus-System with S7-Master.
//The call of the diagnostic block must be made in the execution levels 
//OB1, OB82 and OB86. The number of the instance block is freely selectable.
//The call of the Diagnostic-FB must be the same in all execution levels 
//(DB number, list of parameters).
//All interrupts are delayed during execution of the function block. 
//
AUTHOR : SIEMENS
FAMILY : DP
NAME : Diagnose
VERSION : 4.5
VAR_INPUT
  DP_MASTERSYSTEM : INT  := 1;	//DP_Mastersystem-Nr.
  EXTERNAL_DP_INTERFACE : BOOL ;	//Externe DP-Schnittstelle (CP/IM)
  MANUAL_MODE : BOOL ;	//Betriebsart Hand fuer Einzeldiagnose
  SINGLE_STEP_SLAVE : BOOL ;	//Durchwahl der DP_Slaves
  SINGLE_STEP_ERROR : BOOL ;	//Durchwahl der Fehler auf dem DP_Slave
  RESET : BOOL ;	//Auswertung zuruecksetzen
  SINGLE_DIAG : BOOL ;	//DP_Slave-Einzeldiagnose
  SINGLE_DIAG_ADR : BYTE ;	//DP_Slave-Adresse bei Einzeldiagnose
END_VAR
VAR_OUTPUT
  ALL_DP_SLAVES_OK : BOOL  := TRUE;	//Alle DP-Slaves sind o.k.
  SUM_SLAVES_DIAG : BYTE ;	//Anzahl der betroffenen Slaves
  SLAVE_ADR : BYTE ;	//DP_Slave-Adresse
  SLAVE_STATE : BYTE ;	//0:o.k., 1:ausgefallen, 2:gestoert, 3:nicht projektiert/nicht auswertbar
  SLAVE_IDENT_NO : WORD ;	//Ident-Nummer des DP-Slaves
  ERROR_NO : BYTE ;	//Fehler-Nummer
  ERROR_TYPE : BYTE ;	//1:Slotdiag, 2:Modulstatus, 3:Kanaldiag, 4:S7-Diag, 5:Geratediag, 6:Leitungsdiag
  MODULE_NO : BYTE ;	//Modul-Nr.
  MODULE_STATE : BYTE ;	//Modul-Status
  CHANNEL_NO : BYTE ;	//Kanal-Nr.
  CHANNEL_TYPE : BYTE ;	//Kanal-Typ
  CHANNEL_ERROR_CODE : INT ;	//Kanal-Fehlercode
  CHANNEL_ERROR_INFO_1 : DWORD ;	//Kanal-Fehlerinformation (Teil 1)
  CHANNEL_ERROR_INFO_2 : DWORD ;	//Kanal-Fehlerinformation (Teil 2)
  DIAG_COUNTER : BYTE ;	//Anzahl der Diagnosen des Slaves
  DIAG_OVERFLOW : BOOL ;	//Diagnoseueberlauf
  BUSY : BOOL ;	//Auswertung laeuft
END_VAR
VAR
  DONE_READ_SZL_092 : BOOL ;	//SZL 092-Lesen abgeschlossen
  DONE_READ_SZL_292 : BOOL ;	//SZL 292-Lesen abgeschlossen
  DONE_READ_SZL_692 : BOOL ;	//SZL 692-Lesen abgeschlossen
  SZL692_NOT_SUPP : BOOL ;	//SZL 692-Lesen nicht moeglich
  START_END : BOOL ;	//Anlauf abgeschlossen
  NEW_SLAVE_DIAG : BOOL ;	//Neue Dignose des Slaves liegt vor
  SAME_SLAVE_DIAG : BOOL ;	//Neue Diagnose vom angezeigten Slave
  SFC13_ACTIV : BOOL ;	//SFC13-Lesen aktiv
  SZL_C91_ACTIV : BOOL ;	//SZLC91-Lesen aktiv
  SINGLE_DIAG_ACTIV : BOOL ;	//Einzeldiagnose aktiv
  NEXT_REQUEST : BOOL ;	//Folgeauftraege in ULL vorhanden
  EDGE_TIPP_SLV : BOOL ;	//Flankenmerker bei Slave_Tippen
  EDGE_TIPP_ERR : BOOL ;	//Flankenmerker bei Fehler_Tippen
  EDGE_RESET : BOOL ;	//Flankenmerker bei Reset
  EDGE_SINGLE_DIAG : BOOL ;	//Flankenmerker bei Einzeldiagnose
  INCH_SLV_START : BOOL ;	//Slave_Tippen: Erstmaliges Slave-Tippen
  INCH_ERR_START : BOOL ;	//Error_Tippen: Erstmaliges Error-Tippen
  DIAG_BLOCK_START : BOOL ;	//Error_Tippen: Start Diagnoseblockauswertung
  SRCH_FIRST_START : BOOL ;	//Betroffenen Slave suchen: Erstmaliges Suchen
  RESET_DIAG : BOOL ;	//Diagnoseauswertung ruecksetzen
  PARAM_ERROR : BOOL ;	//Parametrierfehler
  BUSY_SFC : BOOL ;	//Busy bei SFC-Bearbeitung
  BIE_OK : BOOL ;	//BIE-Bit
  SLOT_DIAG_EXIST : BOOL ;	//Kennungsdiagnose vorhanden
  CHANNEL_DIAG_EXIST : BOOL ;	//Kanaldiagnose vorhanden
  S7_DIAG_ALARM : BOOL ;	//S7-Slave mit Diagnosealarm vorhanden
  S7_DIAG_EXIST : BOOL ;	//S7-Diagnose (DS0/1) vorhanden
  NO_DIAG_INFO_EXIST : BOOL ;	//Keine Diagnoseinfo vorhanden
  NO_DPV1_SLOT_MODEL : BOOL ;	//Kein DPV1-Slotmodell vorhanden
  SUM_SLAVES_DIAG_INT : BYTE ;	//Anzahl der betroffenen Slaves (gesichert)
  RESERVE_BYTE : BYTE ;	//Reserve-Byte
  TIPP_SLV_INDEX : DWORD ;	//Slave_Tippen: Adresse des Akt. Slaves
  TIPP_ERR_INDEX : DWORD ;	//Error_Tippen: Adresse des Akt. Fehlers
  DIAG_LOG_ADDR : WORD ;	//Diagnose/Logische-Adresse des Slaves
  DIAG_LEN_SFC13 : BYTE ;	//Von SFC13 gelieferte Laenge der Diagnosedaten inkl.Header
  ACT_DIAG_LEN : BYTE ;	//Aktuelle Gesamtlaenge der Diagnose
  DIAG_BLOCK_LEN : BYTE ;	//Laenge des aktuellen Diagnosebocks
  HEADER_IDENT : BYTE ;	//Diagnosekennung im Header
  DIAG_BLOCK_INDEX_CNT : BYTE ;	//Pruefzaehler im Diagnoseblock
  ERROR_NR : BYTE ;	//Fehlernummer
  SLAVE_ADDRESS : WORD ;	//Nummer des betroffenen Slaves
  START_ADR_BLOCK : DWORD ;	//Startadresse des Diagnoseblocks
  WRITE_INDEX : INT ;	//Position: aktueller Schreibzeiger
  READ_INDEX : INT ;	//Position: aktueller Lesezeiger
  WRITE_CNT : INT ;	//Schreibzaehler: Anzahl der Diagnosen
  POLLING_LIST_ADR : ARRAY  [1 .. 32 ] OF //Umlaufliste fuer Diag-/Log.Baseadressen
  WORD ;
  SLAVE_SLOTS : ARRAY  [1 .. 756 ] OF //48 Slots pro Slave (126 x 6 Byte)
  BYTE ;
  TOP_SI : STRUCT 	//Lokaldaten Aktueller OB
   EV_CLASS : BYTE ;
   EV_NUM : BYTE ;
   PRIORITY : BYTE ;
   NUM : BYTE ;
   TYP2_3 : BYTE ;
   TYP1 : BYTE ;
   ZI1 : WORD ;
   ZI2_3 : DWORD ;
  END_STRUCT ;
  SZL_READ_C91 : ARRAY  [1 .. 16 ] OF //Datenfach fuer SZL C91-Daten
  BYTE ;
  ACT_DAT : ARRAY  [1 .. 22 ] OF //Aktuelles Datenfach
  BYTE ;
  DIAG_DAT_NORM : ARRAY  [1 .. 244 ] OF //Slave-Diagnosedaten
  BYTE ;
  CONFIG_SLAVES : ARRAY  [1 .. 4 ] OF //Projektierte Slaves
  DWORD ;
  EXIST_SLAVES : ARRAY  [1 .. 4 ] OF //Ansprechbare Slaves
  DWORD ;
  FAILED_SLAVES : ARRAY  [1 .. 4 ] OF //Ausgefallene Slaves
  DWORD ;
  FAULTY_SLAVES : ARRAY  [1 .. 4 ] OF //Gestoerte Slaves
  DWORD ;
  AFFECT_SLAVES : ARRAY  [1 .. 4 ] OF //Betroffene Slaves (ausgefallen oder gestoert)
  DWORD ;
  AFFECT_SLAVES_MEM : ARRAY  [1 .. 4 ] OF //Betroffene Slaves gespeichert (ausgefallen oder gestoert)
  DWORD ;
  DIAG_CNT : ARRAY  [1 .. 126 ] OF //Anzahl der Diagnosen pro Slave
  BYTE ;
  RESERVE : WORD ;	//Reserve-Byte
  DP_MASTERSYSTEM_INT : INT  := 1;	//DP_Mastersystem-Nr. (intern)
  EXT_DP_INTERFACE_INT : BOOL ;	//Externe DP-Schnittstelle (intern)
  MANUAL_MODE_INT : BOOL ;	//Handbetrieb (intern)
  SINGLE_STEP_SLAVE_INT : BOOL ;	//Slave-Tippen (intern)
  SINGLE_STEP_ERROR_INT : BOOL ;	//Fehler-Tippen (intern)
  RESET_INT : BOOL ;	//Reset (intern)
  SINGLE_DIAG_INT : BOOL ;	//Einzel-Diagnose (intern)
  CONTROL_INT : BOOL ;	//Funktions-Steuerung intern
  RESERVE_BIT : BOOL ;	//Reserve-Bit (intern)
  SINGLE_DIAG_ADR_INT : BYTE ;	//Slave fuer Einzeldiagnose (intern)
END_VAR
VAR_TEMP
  MAST_SYSTEM_ID : WORD ;	//Nummer des DP-Mastersytems
  LOOP_CNT_1 : INT ;	//Schleifenzaehler 1
  LOOP_CNT_2 : INT ;	//Schleifenzaehler 2
  TEMP_VAR_1 : DWORD ;	//Arbeitsvariable 1
  TEMP_VAR_2 : DWORD ;	//Arbeitsvariable 2
  RETVAL_SFC : INT ;	//RETVAL der SFCs
  SZL_ID : WORD ;	//SZL-ID bei SFC51-Bearbeitung
  SZL_HEADER : STRUCT 	//SZL-Header bei SFC51-Bearbeitung
   LENGHTDR : WORD ;
   N_DR : WORD ;
  END_STRUCT ;
  MDL_ADDR : WORD ;	//MDL-Adresse
  DIAG_ADDR : WORD ;	//DIAG-Adresse
  IO_FLAG : BYTE ;	//IO_FLAG
  SUBNET_ID : BYTE ;	//Subnet-ID
  SLAVE_SFC49_5 : WORD ;	//Slave-Nr.
  SLOT_SFC49_5 : WORD ;	//Steckplatz-Nr.
  ADDR_SFC49_5 : WORD ;	//Offset im Adressraum
  AREA_SFC49_5 : BYTE ;	//Bereichskennung
  OFFSET_ULL : BYTE ;	//Offset Umlaufliste
  DP_SS_TYP : WORD ;	//Typ der DP-Schnittstelle
  START_UP_SI : STRUCT 	//Lokaldaten Anlauf-OB
   EV_CLASS : BYTE ;
   EV_NUM : BYTE ;
   PRIORITY : BYTE ;
   NUM : BYTE ;
   TYP2_3 : BYTE ;
   TYP1 : BYTE ;
   ZI1 : WORD ;
   ZI2_3 : DWORD ;
  END_STRUCT ;
END_VAR
BEGIN
NETWORK
TITLE = Interrupts verzoegern, BUSY-Bit setzen 
//Author: Ralph Buesgen, A&D AS SM7
//V1.0: 03.07.1999: Erstellung des Diagnose-FB
//V1.1: 08.07.1999: Optimierung der Auswertemechanismen bei Fehler-Tippen         
//V2.0: 12.07.1999: Einzeldiagnose von Slaves
//V2.0: 22.07.1999: Auswertung von DS1 als geraetebezogene Diagnose bei 
//                  Siemens-Slaves mit PNO_ID =80xx
//V2.1: 02.08.1999: OB-Lokaldaten mit SFC6 lesen und auswerten
//                  Fehlerauswertung auch bei ausgefallenen Slaves
//V2.2: 14.08.1999: Umlauflistenverwaltung bei Diagnosen im OB82
//V2.3: 31.08.1999: Fehlerbereinigung Kennungsdiagnose bei Stationsausfall
//V2.4: 16.09.1999: Fehlerbereinigung Mastersystem_ID-Abrage bei Anzahl DP-SS >1
//                  Optimierung Diagnose-Erkennung bei OB82 
//                  Erweiterung der Fehlerinfos durch DS0-Bits
//                  Unterscheidung zwischen DS0- und DS1-Auswertung 
//V2.5: 19.09.1999: OB82-Bearbeitung mit SFC5-Lesen und erweiterte Auswertung 
//                  der BGZDs (SZL C91-Daten)
//V2.6: 25.09.1999: Einfuehrung von Bitleisten (48 Bits) fuer die Slots pro Slave 
//                  48 Slots koennen maximal bei S7-Slaves projektiert werden.
//                  Gestoert-Zustand des Slaves ist abhaengig von gest. Slots
//                  Bei Normslave-Diagnose wird immer Slot 2 als Stellvertreter   
//                  gemeldet.
//V2.7: 30.09.1999: Auswertungserweiterung im OB82 bei Slave_Nr.=0 im C91-Fach
//                  Auswertungserweiterung im OB86 bei Wiederkehr des DP-Slaves
//V2.7: 02.10.1999: Verbesserte Auswertung des Parametrierfehlers
//V2.8: 05.10.1999: Fehlerbereinigung bei Einzeldiagnose
//V3.0: 05.10.1999: identisch mit V2.8 -> offizieller Stand fuer die Kunden
//V3.1: 09.10.1999: Erweiterung der Bitleisten um Betr_Slaves_Mem, d.h.
//                  Speichern der betroffenen Slaves bis zum Neustart oder Reset
//V3.2: 12.10.1999: Erweiterung der Fehlerinfos bei S7-Slaves durch DS0 ueber
//                  Ausgangsparameter SPEZIAL_ERROR_INFO  
//V3.3: 17.10.1999: Slave-Status "ausgefallen" bei "Diag_Deactivated"
//                  Im Anlauf/Reset kein Loeschen der Bitleiste Betr_Slaves_Mem
//V3.3: 17.01.2000: Fehlertyp "Allgemeine Geraetediagnose" eingefuehrt ohne
//                  spezielle Zusatzinfos
//V3.3: 01.02.2000: BIE-Bit setzen
//V3.4: 07.07.2000: Im aktuellen Fach wird unter "KANALTYP" eingetragen
//                  bei Norm-Kanal: 01=Eingabe, 02=Ausgabe, 03=Ein/Ausgabe
//                  bei S7-Kanal: 70=DI, 71=AI, 72=DO, 73=AO, 74=FM_POS... 
//V3.4: 15.07.2000: Neuer Ausgangsparameter "CHANNEL_TYP" 
//V3.4: 18.07.2000: Bitgranulare Peripherie aus DS1 in "CHANNEL_ERROR_INFO" 
//                  kopieren (z.B. ASI-CP mit max. 32 ASI-Slaves)
//V3.4: 20.07.2000: Bei neuem ASI-CP mit 64 Slaves werden in "SPEZIAL_ERROR_INFO"
//                  die restlichen 32 Slaves abgelegt. DS0-Inhalt wird somit
//                  ueberschrieben. 
//V3.4: 24.07.2000: Wenn neben Kennungsdiagnose noch andere Diagnosebloecke 
//                  vorliegen, dann wird Kennungsdiagnose nicht ausgewertet.
//V3.4: 28.07.2000: Bei Hand-Einzeldiagnose "immer" Diagnoseauswertung
//V3.4: 04.08.2000: Jedem Kanal-Fehler (Norm- und S7) wird ein eindeutiger 
//                  Fehler-Code zugeordnet. 
//                  Erweiterung aktuelles Fach durch Wortfeld "Error-Code".
//                  Neuer Ausgangsparameter "CHANNEL_ERROR_CODE".  
//V3.4: 08.08.2000: Umbenennung "SPEZIAL_ERROR_INFO" in "CHANNEL_ERROR_INFO_2".   
//V3.5: 18.08.2000: Diagnosen pro Slave zaehlen (OB86/OB82 kommend+gehend).
//                  Neuer Ausgangsparameter "DIAG_COUNTER".
//                  Kanalfehler ueber Potenzieren (2^Error_Code) bitcodiert,
//                  keine Sprungleiste wie bisher.
//V3.5: 09.09.2000: Fehlerumgehung, wenn SZL C91 in OB82 nicht lesbar.
//                  In diesem Falle wird im OB1 der Leseversuch neu gestartet. 
//                  Zwischenspeicherung "Summe betroffenen Slaves". Erst am 
//                  FB-Ende erfolgt die Uebergabe an den Ausgangsparameter. 
//                  Zu Beginn werden die Eingangsparameter gesichert (aus 
//                  Konsistenzgruenden) und mit gesicherten Werten gearbeitet
//V3.5: 15.09.2000: 32-Bit-Pruefung im CHANNEL_ERROR_CODE, frueher nur 16-Bit
//V3.5: 16.09.2000: Code fuer Geraetediagnose nur dann ausgeben, wenn Slave  
//                  betroffen oder S7-Slave.
//V3.5: 21.09.2000: Loeschen der Bitleisten Proj-, Vorh- und Betr-Slaves in der 
//                  RESET-Routine.
//V3.5: 22.09.2000: Funktionssteuerung ueber DB-Bit "CONTROL_INT", d.h. entweder
//                  ueber Einlesen der Eingangsparameter oder direkt ueber die
//                  internen Variablen.   
//V3.5: 27.09.2000: Optimierung in der Anlauf/Reset-Routine bei SZLx92-Lesen 
//V4.0: 29.09.2000: Umbennung V3.5 -> V4.0
//V4.1: 13.10.2000: Fehlerbereinigung, wenn SZL C91-Lesen und SFC13-Bearbeitung   
//                  durch neuen Diagnosealarme unterbrochen werden.
//                  Im aktuellen Fach wird in Byte 6+7 die Diagnoseadresse des
//                  Slaves abgelegt. 
//V4.1: 20.10.2000: Neue Temp-Variable DIAG_ADDR (neben MDL_ADDR), die eine 
//                  getrennte Ablage der MDL- und Diag-Adresse ermoeglicht.  
//V4.1: 04.11.2000: Besteht die Gesamtdiagnose neben der Kennungsdiagnose aus 
//                  weiteren Diagnosebloecken, erfolgt keine Auswertung der 
//                  Kennungsdiagnose. Wenn in der S7-Geraetediagnose (DS0/1)      
//                  aber keine Infos stehen, wird die anfaenglich uebersprungene  
//                  Kennungsdiagnose erneut ausgewertet.  
//V4.2: 23.12.2000: Einbindung Diagnoserepeater  
//V4.2: 18.04.2001: Einbindung Diagnoserepeater  
//V4.2: 19.04.2001: Einbindung Diagnoserepeater
//V4.3: 05.12.2001: DPV1-Integration 
//                  am SFC5 Slot=2 bei S7-Slotmodell anparametriert
//                  am SFC5 Slot=0 bei V1-Slotmodell anparametriert
//V4.4: 28.06.2002: Fehlerbereiningung. Ermitteln Slavesadresse aus dem Tippindex 
//                  im Tippbetrieb. Initialisierung der Slaveadresse, wenn alle 
//                  Slaves o.k. 
//V4.5: 04.12.2002: Erweiterung der DS1-Auswertung (8 <= DS1 <= 48).
//
      CALL  "DIS_AIRT" (
           RET_VAL                  := #RETVAL_SFC);	//Interrupts verzoegern
      SET;
      S     DIX 27.1;	//FB-Bearbeitung starten
      S     DIX 30.6;	//BIE-Bit setzen
      A     DIX 1402.6;	//Wenn Interne Steuerung aktiv
      JC    EXT1;	//-> keine Eingangsparameter einlesen
      L     DIW 0;	//DP-Mastersystem_Nr lesen
      T     DIW 1400;	//und sichern
      L     DIB 3;	//Adresse fuer Einzeldiagnose lesen
      T     DIB 1403;	//und sichern
      A     DIX 2.0;	//Bit-Eingangsparameter lesen
      =     DIX 1402.0;	//und sichern
      A     DIX 2.1;
      =     DIX 1402.1;
      A     DIX 2.2;
      =     DIX 1402.2;
      A     DIX 2.3;
      =     DIX 1402.3;
      A     DIX 2.4;
      =     DIX 1402.4;
      A     DIX 2.5;
      =     DIX 1402.5;
EXT1: L     DIW 1400;	//Gesichertes DP-Mastersystem
      T     #MAST_SYSTEM_ID;	//intern speichern
      T     #SUBNET_ID;
      L     P##POLLING_LIST_ADR;	//Startadresse 1. ULL-Fach
      SLD   8;	//Bereichskennung loeschen
      SRD   11;	//Bitnummer loeschen
      T     #OFFSET_ULL;	//-> temp. sichern
NETWORK
TITLE = Welcher OB wird aktuell bearbeitet?
//Mit dem SFC6 werden die Lokaldaten des aktuell bearbeiteten OBs gelesen.
//Aus den Startinfos des aufrufenden OBs wird die Nummer des aktuell bearbeiteten 
//OBs ausgelesen, von dem aus der Diagnose-FB aufgerufen wird. Entsprechend wird 
//in die Bearbeite-Routine verzweigt.
      BLD   7;	//Lokaldaten des aktuellen OBs lesen
      L     DINO;
      T     LW 50;
      L     P#DBX 882.0;
      T     LD 52;	//Wenn Fehler bei SFC6-Bearbeitung
      L     0;	//-> BIE-Bit ruecksetzen
      T     LW 56;	//-> Ende Baustein
      L     P#V 38.0;	//Startadresse Lokaldaten
      T     LD 58;	//OB_NUMBER: 1 
      UC    "RD_SINFO";	//Aktuelle OB_Nr.
      {     P#L 14.0, P#L 50.0, P#L 56.0 };
      BLD   8;
      AN    BR;	//OB_NUMBER: 82 
      R     DIX 30.6;
      JC    ENDE;
      LAR1  P##TOP_SI;
      L     B#16#1;	//OB_NUMBER: 86 
      L     DIB [AR1,P#3.0];
      ==I;
      JC    OB1;	//Andere OBs werden nicht unterstuetzt
      L     B#16#52;
      ==I;
      JC    OB82;
      TAK;
      L     B#16#56;
      ==I;
      JC    OB86;
      JU    ENDE;
NETWORK
TITLE = Ausfall eines Slaves (nur OB86)
//Es wird geprueft, ob der OB86-Aufruf von der dezentralen Peripherie ausgeloest 
//wurde. Aus den Startinfos des OB86 wird die Mastersystem-ID und die Slave-Nr. 
//ausgewertet und in das C91-Fach eingetragen. Die ermittelte Slave_Nr. wird in 
//die Bitleisten Vorh_Slaves, Ausgef_Slaves, Betr_Slaves und Betr_Slaves_Mem 
//ein- bzw. ausgetragen. Die Anzahl der Diagnosen des gemeldeten Slaves wird
//inkrementieren. 
OB86: LAR1  P##TOP_SI;	//Startadresse Lokaldaten
      A(;
      L     DIB [AR1,P#1.0];
      L     B#16#C4;	//Wenn Fehlercode "Ausfall DP-Station"
      ==I;
      );
      O(;
      TAK;
      L     B#16#C5;	//Wenn Fehlercode "Stoerung DP-Station"
      ==I;
      );
      O(;
      TAK;
      L     B#16#C7;	//Wenn Fehlercode "Wiederkehr DP-Station"
      ==I;	//aber mit Baugruppen-Parametrierfehler
      );
      O(;
      TAK;
      L     B#16#C8;	//Wenn Fehlercode "Wiederkehr DP-Station"
      ==I;	//aber mit Abweichung Soll-/Istausbau
      );	//-> dezentraler Ausfall/Wiederkehr
      JCN   ENDE;	//sonst zentral -> Ende Baustein
//Pruefen, ob gemeldetes und anparametriertes Mastersystem identisch.
      L     DIB [AR1,P#10.0];	//Wenn Mastersystem-ID aus Lokaldaten
      L     #MAST_SYSTEM_ID;	//nicht identisch mit Eingangsparameter
      <>I;
      =     DIX 30.4;	//-> Parametrierfehler
      JC    ENDE;	//-> Ende Baustein
      L     DIB [AR1,P#11.0];	//Wenn Slave_Nr. aus Lokaldaten =0
      L     0;
      ==I;
      =     DIX 30.4;	//-> Parametrierfehler
      JC    ENDE;	//-> Ende Baustein
      S     DIX 28.5;	//sonst NEW_SLAVE_DIAG-Bit setzen
      LAR2  P##ACT_DAT;	//Startadresse aktuelles Fach
      L     DIB [AR2,P#0.0];	//Wenn aktuell angezeigter Slave
      L     DIB [AR1,P#11.0];	//gleich dem neu gemeldeten Slave
      ==I;
      S     DIX 28.6;	//-> SAME_SLAVE_DIAG-Bit setzen
      LAR2  P##SZL_READ_C91;	//Startadresse C91-Fach (BGZD)
      L     DIW [AR1,P#10.0];	//Mastersystem-ID und Slave_Nr.
      T     #DP_MASTERSYSTEM;	//in C91-Fach eintragen
      L     DW#16#0;
      T     DIW [AR2,P#2.0];	//Restliches C91-Fach loeschen
      T     DID [AR2,P#4.0];
      T     DID [AR2,P#8.0];
      T     DID [AR2,P#12.0];
//Anzahl der Diagnosen des Slaves inkrementieren.
      L     DIB [AR1,P#11.0];	//Slave_Nr. aus Startinfo OB86
      DEC   1;	//Slaveposition = Slave_Nr.-1
      SLD   3;	//Byteadresse
      L     P##DIAG_CNT;	//+ Startadresse Diagnose_Zaehler  
      +D;
      LAR2;	//-> Position Diagzaehler des Slaves 
      L     DIB [AR2,P#0.0];	//Diagnoseanzahl inkrementieren
      INC   1;
      T     DIB [AR2,P#0.0];
//Slave_Nr. in Bitleisten ein- bzw. austragen. 
      L     DIB [AR1,P#11.0];	//Slave_Nr. aus Startinfo OB86
      L     8;	//:8 -> Akku1-L (Byteadresse) 
      /I;
      T     #TEMP_VAR_1;	//   -> Akku1-H (Bitadresse)
      AD    DW#16#FFFF;
      T     #TEMP_VAR_2;	//Byte-Nr. sichern
      L     DW#16#0;
      L     #TEMP_VAR_1;
      SRD   16;	//Bitadresse ermitteln
      <>D;	//Wenn Bitadresse <>0
      JC    GAN1;	//-> Bitadresse sofort dekrementieren
      L     B#16#8;	//sonst Bitadr.=8 -> spaeter dekrement.
      T     #TEMP_VAR_1;	//sichern
      L     #TEMP_VAR_2;
      DEC   1;	//Byte-Nr. dekrementieren
      T     #TEMP_VAR_2;
      TAK;
GAN1: DEC   1;	//Bitadresse dekrementieren
      L     #TEMP_VAR_2;
      SLD   3;	//Byteadresse
      +D;	//+ Bitadresse -> Neue Slaveposition
      L     P##EXIST_SLAVES;	//+ Offset Bitleiste Vorh_Slaves
      +D;
      LAR2;	//-> Slavepos. in Bitleiste Vorh_Slaves
      A     DIX [AR1,P#0.0];	//EV_CLASS: Slaveausfall/Wiederkehr
//Stationsausfall
      R     DIX [AR2,P#0.0];	//-> Slave nicht mehr vorhanden
      S     DIX [AR2,P#16.0];	//-> Slave ausgefallen
      S     DIX [AR2,P#48.0];	//-> Slave betroffen
      S     DIX [AR2,P#64.0];	//-> Slave betroffen speichern
      R     DIX [AR2,P#32.0];	//-> Slave nicht mehr gestoert 
      JC    ENDE;	//-> Ende Baustein
//Stationswiederkehr
      S     DIX [AR2,P#0.0];	//-> Slave wieder vorhanden
      R     DIX [AR2,P#16.0];	//-> Slave nicht mehr ausgefallen
      AN    DIX [AR2,P#32.0];	//Wenn Slave zus. nicht gestoert
      R     DIX [AR2,P#48.0];	//-> Slave nicht mehr betroffen
      JU    ENDE;	//-> Ende Baustein
NETWORK
TITLE = Stoerung eines Slaves (nur OB82)
//Aus den Startinfos des OB82 wird die Diagnoseadresse/Logische Basisadresse des 
//gestoerten Slaves ermittelt. Es wird ueber SFC49 geprueft, ob die Diagnose vom 
//dezentralen Bereich kommt. Ob der Slave gestoert ist, wird ermittelt ueber die 
//Anzahl der gestoerten Slots pro Slave. Sind keine gestoerten Slots fuer den 
//gemeldeten Slave eingetragen, gilt der Slave als nicht_gestoert. Fuer jeden 
//Slave werden 48 Slots reserviert. Diese Zahl ergibt sich aus 5 Byte-SKF-Format 
//bei S7-Slaves in einem 244-Byte-Konfigtelegramm. Bei Normslaves meldet immer 
//Slot 2 als Stellvertreter die Diagnose. 
//Fuer die Ermittlung Mastersystem-ID, Slave-Nr. und Baugruppenstatus wird die 
//SZL C91 mit SFC51 gelesen. Bei externen DP-Schnittstellen (CP/IM) laeuft das 
//lesen der SZL C91 asynchron. Deshalb wird eine Umlaufliste verwendet, damit 
//die waehrend der OB82-Bearbeitung eintreffenden Diagnosen nicht verloren gehen. 
//Bei eintreffenden Diagnosen wird ein Schreibezeiger, bei der Abarbeitung der 
//Diagnoseeintraege ein Lesezeiger verwendet. Die Umlaufliste hat Platz fuer 
//max. 32 Eintraege. Ein Schreibzaehler ueberwacht die Anzahl der ULL-Eintraege.
//Die ermittelte Slave-Nr. wird in die Bitleisten Gestoe_Slaves, Ausgef_Slaves, 
//Betr_Slaves und Betr_Slaves_Mem ein- bzw. ausgetragen. Die Anzahl der Diagnosen
//des gemeldeten Slaves wird inkrementiert.
OB82: LAR1  P##TOP_SI;	//Startadresse Lokaldaten
      L     DIB [AR1,P#5.0];	//OB82_IO_FLAG
      T     #IO_FLAG;	//Eing.=54H, Ausg.=55H 
      L     DIW [AR1,P#6.0];	//OB82_MDL_ADR
      T     #MDL_ADDR;	//temp. sichern
//Abfrage, ob Diagnose vom DP-Bereich kommt.
      CALL  "LGC_GADR" (
           IOID                     := #IO_FLAG,
           LADDR                    := #MDL_ADDR,
           RET_VAL                  := #RETVAL_SFC,
           AREA                     := #AREA_SFC49_5,
           RACK                     := #SLAVE_SFC49_5,
           SLOT                     := #SLOT_SFC49_5,
           SUBADDR                  := #ADDR_SFC49_5);	//Slave logisch -> geografisch / Eingangs- bzw. Ausgangskennung / log. Base-/Diagadr. / Bereichskennung / Slave_Nr. / Steckplatz / Subaddr
      AN    BR;	//Wenn Fehler bei SFC49-Bearbeitung
      R     DIX 30.6;	//-> BIE-Bit ruecksetzen
      JC    ENDE;	//-> Ende Baustein
      L     #AREA_SFC49_5;	//Bereichskennung auswerten
      L     B#16#2;	//Kennung fuer DP =2
      <>I;
      JC    ENDE;	//Wenn keine DP-Kennung -> Ende
      L     DIW 60;	//Wenn Umlaufliste voll
      L     32;
      ==I;
      S     DIX 27.0;	//-> Diagnoseueberlauf
      JC    ENDE;	//-> Ende Baustein
//Schreibezeiger inkrementieren und Diagnose-/Log.Baseadresse in ULL eintragen.
//Solange SZL_C91-Lesen aktiv ist, wird kein ULL-Fach abgearbeitet.
//Bei Eintreffen einer Diagnose wird ein Auftrags-Merker gesetzt.
      L     DIW 60;	//Anzahl der Diagnosen inkrementieren
      +     1;
      T     DIW 60;
      L     0;	//Wenn Anzahl der Diagnosen >0
      >I;
      =     DIX 29.2;	//-> (Folge-)Auftrag liegt vor
      L     DIW 56;	//Schreibezeiger +1
      +     1;
      L     32;	//Und (Max_Anzahl -1)
      +     -1;
      AW;
      T     DIW 56;	//-> neuer Schreibezeiger
      L     2;	//* Groesse ULL-Fach (1 Wort)
      *I;
      L     #OFFSET_ULL;	//+ Startoffset ULL
      +I;
      SLD   3;
      LAR2;	//-> Adresse neues ULL-Fach
      AN    DIX [AR1,P#5.0];	//Wenn Ausgabebaugruppe
      L     #MDL_ADDR;
      JC    DADR;
      OW    W#16#8000;	//-> A-Bit in Adresse setzen
DADR: T     #DP_MASTERSYSTEM;	//und in neues ULL-Fach eintragen
      A     DIX 29.0;	//Solange SZL_C91-Lesen aktiv
      JC    ENDE;	//-> Ende Baustein
//Lesezeiger inkrementieren und Diagnose/Log.Baseadresse aus ULL lesen.
//Wenn noch nicht alle ULL-Eintraege bearbeitet sind, wird der
//Auftragsmerker gesetzt.
ULL:  L     DIW 60;	//Anzahl Diagnosen dekrementieren
      +     -1;
      T     DIW 60;
      L     0;	//Wenn Anzahl der Diagnosen >0
      >I;
      =     DIX 29.2;	//-> Folgeauftrag liegt vor
      L     DIW 58;	//Lesezeiger +1
      +     1;
      L     32;	//Und (Max_Anzahl -1)
      +     -1;
      AW;	//-> neuer Lesezeiger
      T     DIW 58;
      L     2;	//* Groesse ULL-Fach (1 Wort)
      *I;
      L     #OFFSET_ULL;	//+ Startoffset ULL
      +I;
      SLD   3;
      LAR2;	//-> Adresse ULL-Fach
      L     #DP_MASTERSYSTEM;	//Diag./Log.-Adresse aus ULL-Fach
      T     DIW 42;
//Bei integrierter DP-SS (CPUs) wird SZL 0C91, bei externer DP-SS (CPs)
//wird SZL 4C91 gelesen. Die Schnittstellen werden unterschieden 
//ueber den Eingangsparameter "EXTERNAL_DP_INTERFACE".
C91:  AN    DIX 1402.0;
      L     W#16#0;	//Typ: Interne DP-Schnittstelle
      JC    INT1;
      L     W#16#4000;	//Typ: Externe DP-Schnittstelle
INT1: T     #DP_SS_TYP;
      OW    W#16#C91;
      T     #SZL_ID;	//Bildung SZL-ID
      BLD   7;	//SZL_C91 (BGZD) lesen
      SET;
      =     L 50.0;
      L     DIW 42;	//Diag./Log.-Adresse
      T     LW 51;
      L     0;
      T     LW 53;
      L     P#V 18.0;	//Datenfach fuer SZL_C91-Daten
//Wenn im OB82 die SZL C91 nicht gelesen werden kann, wird im OB1 "ein" 
//neuer Versuch gestartet, diese SZL zu lesen. Wenn dieser ebenfalls 
//misslingt, dann liegt ein Parametrierfehler vor.
      T     LD 55;	//Startadresse Lokaldaten
      L     W#16#1002;	//Wenn Aktuelle OB_Nr.
      T     LW 59;	//OB_NUMBER: 82 
      L     16;
      T     LW 61;	//und Fehler beim SZL_C91-Lesen 
      L     DINO;	//-> neuer Versuch im OB1-Teil
      T     LW 63;	//Wenn Fehler beim SZL_C91-Lesen 
      L     P#DBX 894.0;	//-> Parametrierfehler
      T     LD 65;	//-> SZL_C91_Lesen deaktivieren
      UC    "RDSYSST";	//-> BIE-Bit ruecksetzen
      {     P#L 50.0, P#L 16.0, P#L 51.0, P#L 14.0, P#L 50.1, P#L 53.0, P#L 59.0 };	//-> Ende Baustein
      A     L 50.1;	//Wenn SZL_C91-Lesen fertig
      =     DIX 30.5;	//-> SZL_C91-Lesen deaktivieren
      BLD   8;	//-> gelesene Daten auswerten
      LAR1  P##TOP_SI;	//sonst SZL_C91-Lesen aktiv 
      L     DIB [AR1,P#3.0];	//-> Ende Baustein
//Pruefen, ob gemeldetes und anparametriertes Mastersystem identisch.
      L     B#16#52;	//Startadresse C91-Fach (BGZD)
      ==I;	//Wenn Mastersystem-ID aus C91-Fach
      AN    BR;	//nicht identisch mit Eingangsparameter
      JC    NEU1;
      AN    BR;	//-> Parametrierfehler
      =     DIX 30.4;	//-> Ende Baustein
      R     DIX 29.0;	//Wenn Slave_Nr. aus C91-Fach =0
      R     DIX 30.6;
      JC    ENDE;
      AN    DIX 30.5;	//-> Parametrierfehler
      R     DIX 29.0;	//-> Ende Baustein
      JC    WAUS;	//sonst NEW_SLAVE_DIAG-Bit setzen
NEU1: S     DIX 29.0;	//Startadresse aktuelles Faches
      JU    ENDE;	//Wenn aktuell angezeigter Slave
WAUS: LAR1  P##SZL_READ_C91;	//gleich dem neu gemeldeten Slave
      L     DIB [AR1,P#0.0];
      L     #MAST_SYSTEM_ID;	//-> SAME_SLAVE_DIAG-Bit setzen
//Steckplatz-Status in Slotleiste des Slaves eintragen.
      <>I;	//Steckplatz aus C91-Fach
      =     DIX 30.4;	//: 8 
      JC    ENDE;	//-> Akku1-L (Byteadresse) 
      L     DIB [AR1,P#1.0];	//-> Akku1-H (Bitadresse)
      L     0;
      ==I;	//Byte-Nr. sichern
      =     DIX 30.4;
      JC    ENDE;
      S     DIX 28.5;	//Bitadresse ermitteln
      LAR2  P##ACT_DAT;	//Wenn Bitadresse <>0
      L     DIB [AR2,P#0.0];	//-> Bitadresse sofort dekrementieren
      L     DIB [AR1,P#1.0];	//Wenn Steckplatz aus C91-Fach =0
      ==I;	//-> neues DPV1-Slotmodell
      S     DIX 28.6;
      L     DIB [AR1,P#2.0];
      L     8;	//-> Slotposition im Slave =0
      /I;	//sonst Bitadr.=8 -> spaeter dekrement.
      T     #TEMP_VAR_1;	//sichern
      AD    DW#16#FFFF;
      T     #TEMP_VAR_2;	//Byte-Nr. dekrementieren
      L     DW#16#0;
      L     #TEMP_VAR_1;
      SRD   16;	//Bitadresse dekrementieren
      <>D;
      JC    GAN2;	//Byteadresse
      L     DIB [AR1,P#2.0];	//+ Bitadresse
      L     B#16#0;	//-> Slotposition im Slave
      T     #TEMP_VAR_1;	//Slave_Nr. aus C91-Fach
      ==I;	//Slaveposition = Slave_Nr.-1
      JC    SLOT;	//sichern
      L     B#16#8;	//* Offset Anzahl Bytes pro Slave
      T     #TEMP_VAR_1;
      L     #TEMP_VAR_2;	//-> Slaveposition
      DEC   1;	//+ Offset Slotposition im Slave
      T     #TEMP_VAR_2;
      TAK;	//+ Offset Startposition 1. Slaveslot
GAN2: DEC   1;
      L     #TEMP_VAR_2;	//-> Absolute Slotposition
      SLD   3;	//Baugruppenzustand = (nicht) gestoert
      +D;	//als Slotstatus eintragen
//Anzahl der Diagnosen des Slaves inkrementieren.
SLOT: T     #TEMP_VAR_2;	//Slaveposition = Slave_Nr.-1
      L     DIB [AR1,P#1.0];	//Byteadresse
      DEC   1;	//+ Startadresse Diagnose_Zaehler  
      T     #TEMP_VAR_1;
      L     6;	//-> Position Diagzaehler des Slaves 
      *I;	//Diagnoseanzahl inkrementieren
      SLD   3;
      L     #TEMP_VAR_2;
//Slave_Nr. in Bitleisten ein- bzw. austragen.
      +D;	//Slave_Nr. aus C91-Fach
      L     P##SLAVE_SLOTS;	//: 8 
      +D;	//-> Akku1-L (Byteadresse) 
      LAR2;	//-> Akku1-H (Bitadresse)
      A     DIX [AR1,P#13.0];
      =     DIX [AR2,P#0.0];	//Byte-Nr. sichern
      L     #TEMP_VAR_1;
      SLD   3;
      L     P##DIAG_CNT;	//Bitadresse ermitteln
      +D;	//Wenn Bitadresse <>0
      LAR2;	//-> Bitadresse sofort dekrementieren
      L     DIB [AR2,P#0.0];	//sonst Bitadr.=8 -> spaeter dekrement.
      INC   1;	//sichern
      T     DIB [AR2,P#0.0];
      L     DIB [AR1,P#1.0];	//Byte-Nr. dekrementieren
      L     8;
      /I;
      T     #TEMP_VAR_1;	//Bitadresse dekrementieren
      AD    DW#16#FFFF;
      T     #TEMP_VAR_2;	//Byteadresse
      L     DW#16#0;	//+ Bitadresse -> Neue Slaveposition
      L     #TEMP_VAR_1;	//+ Offset Bitleiste Ausgef_Slaves
      SRD   16;
      <>D;	//-> Slavepos. in Bitleiste Ausgef_Slaves
      JC    GAN3;	//Slave_Nr. aus C91-Fach
      L     B#16#8;	//Slaveposition = Slave_Nr.-1
      T     #TEMP_VAR_1;	//* Offset Anzahl Bytes pro Slave
      L     #TEMP_VAR_2;
      DEC   1;	//-> Slaveposition
      T     #TEMP_VAR_2;	//+ Offset Startposition 1. Slaveslot
      TAK;
GAN3: DEC   1;	//-> Absolute Slaveposition
      L     #TEMP_VAR_2;	//Wenn Anzahl gestoerte Slots <>0
      SLD   3;
      +D;
      L     P##FAILED_SLAVES;
      +D;
      LAR2;	//-> Slave gestoert
      L     DIB [AR1,P#1.0];
      DEC   1;	//sonst Slave nicht mehr gestoert
      L     6;	//Wenn Slave zus. nicht ausgefallen
      *I;	//-> Slave nicht mehr betroffen
      SLD   3;	//-> Ende Baustein
      L     P##SLAVE_SLOTS;	//-> Slave gestoert
      +D;	//-> Slave betroffen 
      LAR1;	//-> Slave betroffen speichern
      L     DID [AR1,P#0.0];	//-> Ende Baustein
      L     DW#16#0;
      <>D;
      JC    GSTO;
      L     DIW [AR1,P#4.0];
      <>I;
      JC    GSTO;
      R     DIX [AR2,P#16.0];
      AN    DIX [AR2,P#0.0];
      R     DIX [AR2,P#32.0];
      JU    ENDE;
GSTO: S     DIX [AR2,P#16.0];
      S     DIX [AR2,P#32.0];
      S     DIX [AR2,P#48.0];
      JU    ENDE;
NETWORK
TITLE = Initialisierungroutine bei Neustart/Wiederanlauf (nur OB1)
//Im ersten OB1-Zyklus wird die Initialisierung der Variablen durchgefuehrt. 
//Anzahl der ausgefallenen und gestoerten Slaves, das aktuelle Fach, 
//die Adress-Umlaufliste, die Slave-Slots, das SZL C91-Fach, die Faecher der SZLs 
//092/292/692 und die Diagnose-Zaehler werden geloescht. Die Eingangsparameter 
//werden intern gesichert.
OB1:  LAR1  P##TOP_SI;	//Startadresse Lokaldaten
      L     DIB [AR1,P#1.0];	//OB1_SCAN_1: 1=Neu,2=Wieder,3=Zyklus
      L     B#16#2;
      >I;	//Wenn kein Neustart/Wiederanlauf
      JC    ZYKL;	//-> Zyklische Auswertung
//Neu- oder Wiederanlauf, Reset- bzw. Init-Routine
RSET: L     0;	//Initialisieren
      T     DIB 45;	//Gesamtdiagnoselaenge
      T     DIB 46;	//Laenge Diagnoseblock
      T     DID 38;	//Error_Tippindex 
      T     DIB 48;	//Blockauswerte_Index
      T     DIB 49;	//Fehlernummer
      T     DIW 50;	//Slave_Nr.
      T     DIW 56;	//ULL-Schreibzeiger
      T     DIW 58;	//ULL-Lesezeiger
      T     DIW 60;	//ULL-Schreibzaehler
      T     DIB 32;	//Anzahl betroffene Slaves
      L     P##AFFECT_SLAVES;	//Startadr. Bitfeld betr. Slaves 
      T     DID 34;	//-> Slave_Tippindex
      L     P##DIAG_DAT_NORM;	//Startadr. Diagnosefach
      T     DID 38;	//-> Error_Tippindex
      SET;
      R     DIX 28.4;	//Anlaufende ruecksetzen
      R     DIX 28.5;	//Neue Slave-Diagnose ruecksetzen
      R     DIX 28.6;	//Gleiche Slave-Diagnose ruecksetzen
      R     DIX 28.0;	//SZL 092 muss noch gelesen werden
      R     DIX 28.1;	//SZL 292 muss noch gelesen werden
      R     DIX 28.2;	//SZL 692 muss noch gelesen werden
      R     DIX 28.7;	//SFC13-Lesen ruecksetzen
      R     DIX 29.0;	//SZLC91-Lesen ruecksetzen
      R     DIX 29.1;	//Einzeldiagnose ruecksetzen
      R     DIX 29.7;	//Erstmaliges Slave_Tippen
      R     DIX 30.0;	//Erstmaliges Error_Tippen
      R     DIX 30.1;	//Erstmalige Blockauswertung
      R     DIX 30.2;	//Erstmaliges Slave-Suchen
      R     DIX 28.3;	//Fehler bei SZL692-Lesen loeschen
      R     DIX 30.3;	//RESET ruecksetzen
      R     DIX 27.0;	//Diagnoseueberlauf ruecksetzen
      R     DIX 29.2;	//Kein Folgeauftrag
      R     DIX 30.4;	//Parametrierfehler loeschen
      R     DIX 30.7;	//Kennungsdiagnose initialisieren
      R     DIX 31.0;	//Kanaldiagnose initialisieren
      R     DIX 31.1;	//S7-Diagnosealarm initialisieren
      R     DIX 31.2;	//S7-Diagnose initialisieren
      R     DIX 31.4;	//DPV1-Slot-Modell ruecksetzen
      LAR2  P##ACT_DAT;
      L     DW#16#0;	//Aktuelles Fach loeschen
      T     DID [AR2,P#0.0];
      T     DID [AR2,P#4.0];
      T     DID [AR2,P#8.0];
      T     DID [AR2,P#12.0];
      T     DID [AR2,P#16.0];
      T     DIW [AR2,P#20.0];
      LAR1  P##SZL_READ_C91;
      L     #MAST_SYSTEM_ID;	//Eingangsparameter Mastersystem-ID
      T     DIB [AR1,P#0.0];	//in C91-Fach eintragen
      L     DW#16#0;
      T     DIB [AR1,P#1.0];	//Restliches C91-Fach loeschen
      T     DIW [AR1,P#2.0];
      T     DID [AR1,P#4.0];
      T     DID [AR1,P#8.0];
      T     DID [AR1,P#12.0];
      LAR1  P##POLLING_LIST_ADR;	//Alle ULL-Faecher loeschen
      L     16;	//32 ULL-Faecher x 1 Wort/Fach
BLCK: T     #LOOP_CNT_1;	//Anzahl/2 -> 16 Doppelworte
      L     DW#16#0;
      T     DID [AR1,P#0.0];	//ULL-Faecher
      +AR1  P#4.0;
      L     #LOOP_CNT_1;
      LOOP  BLCK;
      LAR1  P##SLAVE_SLOTS;	//Alle Slot-Faecher loeschen
      L     189;	//126 x 6 Bytes/Slave (48 Slots)
DLSL: T     #LOOP_CNT_1;	//Anzahl/4 -> 189 Doppelworte
      L     DW#16#0;
      T     DID [AR1,P#0.0];	//Slot-Faecher
      +AR1  P#4.0;
      L     #LOOP_CNT_1;
      LOOP  DLSL;
      LAR1  P##CONFIG_SLAVES;	//Alle 092/292/692-Faecher loschen
      L     4;	//128 x 1 Bit/Slave = 16 Bytes
SLVS: T     #LOOP_CNT_1;	//Anzahl/4 -> 4 Doppelworte
      L     DW#16#0;
      T     DID [AR1,P#0.0];	//projektierte Slaves
      T     DID [AR1,P#16.0];	//vorhandene Slaves
      T     DID [AR1,P#64.0];	//betroffene Slaves
      +AR1  P#4.0;
      L     #LOOP_CNT_1;
      LOOP  SLVS;
      LAR1  P##DIAG_CNT;	//Alle Diagnose-Zaehler loeschen
      L     32;	//126 x 1 Byte/Slave (+2)
DCNT: T     #LOOP_CNT_1;	//Anzahl/4 -> 32 Doppelworte
      L     DW#16#0;
      T     DID [AR1,P#0.0];	//incl. SLAVE_DIAG_ADR
      +AR1  P#4.0;
      L     #LOOP_CNT_1;
      LOOP  DCNT;
      A     DIX 1402.6;	//Wenn Interne Steuerung aktiv
      JC    EXT2;	//-> keine Eingangsparameter einlesen
      L     DIW 0;	//DP-Mastersystem_Nr lesen
      T     DIW 1400;	//und sichern
      L     DIB 3;	//Adresse fuer Einzeldiagnose lesen
      T     DIB 1403;	//und sichern
      A     DIX 2.0;	//Bit-Eingangsparameter lesen
      =     DIX 1402.0;	//und sichern
      A     DIX 2.1;
      =     DIX 1402.1;
      A     DIX 2.2;
      =     DIX 1402.2;
      A     DIX 2.3;
      =     DIX 1402.3;
      A     DIX 2.4;
      =     DIX 1402.4;
      A     DIX 2.5;
      =     DIX 1402.5;
EXT2: L     DIW 1400;	//Gesichertes DP-Mastersystem_Nr
      T     #MAST_SYSTEM_ID;	//intern speichern
      T     #SUBNET_ID;
      JU    RSZL;	//Starte Lesen SZLs
NETWORK
TITLE = Ermitteln der betroffenen Slaves im Anlauf (nur OB1) 
//Im Anlauf werden die Bitleisten der projektierten, vorhandenen und betroffenen 
//Slaves (gestoert oder ausgefallen) als SZLs (SZL 092/292/692) gelesen. 
//Die betroffenen Slaves werden gespeichert als Betr_Slaves_Mem. Die Bitleisten 
//der ausgefallenen und gestoerten Slaves werden ermittelt. Kann die SZL 692 
//nicht gelesen werden (alter CPU-Stand), werden die ausgefallenen Slaves zu 
//betroffenen Slaves. Ist der Anlauf beendet, wird in den zyklischen Betrieb 
//verzweigt.
ZYKL: A     DIX 28.4;	//Wenn Anlaufbearbeitung abgeschlossen
      JC    AUSW;	//-> Zyklische Auswertung
//Bei integrierter DP-SS (CPUs) wird 0092/0292/0692, bei externer DP-SS
//(CPs) wird 4092/4292/4692 gelesen.
//Die Unterscheidung zwischen interner und externer DP-Schnittstelle (SS)
//erfolgt ueber den Eingangsparameter "EXTERNAL_DP_INTERFACE".
RSZL: AN    DIX 1402.0;
      L     W#16#0;	//Typ: Interne DP-Schnittstelle
      JC    INT2;
      L     W#16#4000;	//Typ: Externe DP-Schnittstelle
INT2: T     #DP_SS_TYP;
      A     DIX 28.0;	//Wenn SZL 092-Lesen fertig
      JC    RDVS;	//-> Pruefe SZL 292-Lesen
      L     #DP_SS_TYP;	//Bildung SZL-ID
      OW    W#16#92;
      T     #SZL_ID;
      BLD   7;	//SZL 092 auslesen = Proj. Slaves
      SET;
      =     L 50.0;
      L     0;
      T     LW 51;
      L     P#V 18.0;
      T     LD 53;
      L     W#16#1002;	//Datenfach fuer SZL092-Daten
      T     LW 57;	//Wenn Fehler beim SZL 092-Lesen
      L     16;	//oder Lesen_fertig (BUSY-Bit =0)
      T     LW 59;	//-> Fertig-Bit setzen
      L     DINO;	//Wenn SZL 292-Lesen fertig
      T     LW 61;	//-> Pruefe SZL 692-Lesen
      L     P#DBX 1176.0;	//Bildung SZL-ID
      T     LD 63;
      UC    "RDSYSST";
      {     P#L 50.0, P#L 16.0, P#L 0.0, P#L 14.0, P#L 50.1, P#L 51.0, P#L 57.0 };	//SZL 292 auslesen = Vorh. Slaves
      A     L 50.1;
      =     DIX 30.5;
      BLD   8;
      AN    BR;
      ON    DIX 30.5;
      S     DIX 28.0;
RDVS: A     DIX 28.1;	//Datenfach fuer SZL292-Daten
      JC    RDBS;	//Wenn Fehler beim SZL 292-Lesen
      L     #DP_SS_TYP;	//oder Lesen_fertig (BUSY-Bit =0)
      OW    W#16#292;	//-> Fertig-Bit setzen
      T     #SZL_ID;	//Wenn SZL 692-Lesen fertig
      BLD   7;	//-> Auswertung aller DONE-Bits 
      SET;	//Bildung SZL-ID
      =     L 50.0;
      L     0;
      T     LW 51;	//SZL 692 auslesen = Betr. Slaves
      L     P#V 18.0;
      T     LD 53;
      L     W#16#1002;
      T     LW 57;
      L     16;
      T     LW 59;
      L     DINO;	//Datenfach fuer SZL692-Daten
      T     LW 61;	//Wenn Fehler beim SZL 692-Lesen
      L     P#DBX 1192.0;	//oder Lesen_fertig (BUSY-Bit =0)
      T     LD 63;	//-> Fertig-Bit setzen
      UC    "RDSYSST";	//Wenn RETVAL=8082
      {     P#L 50.0, P#L 16.0, P#L 0.0, P#L 14.0, P#L 50.1, P#L 51.0, P#L 57.0 };
      A     L 50.1;
      =     DIX 30.5;	//-> SZL692 nicht lesbar (alte CPU)
      BLD   8;	//Solange SZL-Lesen laeuft
      AN    BR;
      ON    DIX 30.5;
      S     DIX 28.1;	//-> Datenausgabe
//Ausgefallene Slaves ermitteln aus Auswertung
//projektierte Slaves exclusiv mit vorhandenen Slaves.
RDBS: A     DIX 28.2;	//Slave ist projektiert =1
      JC    RDCK;	//Slave ist nicht vorhanden =0
      L     #DP_SS_TYP;
      OW    W#16#692;	//-> Slave ist ausgefallen =1
      T     #SZL_ID;
      BLD   7;
      SET;
      =     L 50.0;
      L     0;
      T     LW 51;
      L     P#V 18.0;
      T     LD 53;
      L     W#16#1002;
      T     LW 57;
      L     16;
      T     LW 59;
//Wenn gestoerte Slaves nicht auswertbar:
//Datenfach der gestoerten Slaves loeschen.
//Ausgefallene Slaves werden zu betroffenen Slaves.
//Die betroffenen Slaves werden zusaetzlich gespeichert.
      L     DINO;	//Wenn SZL 692 nicht lesbar
      T     LW 61;
      L     P#DBX 1240.0;
      T     LD 63;	//Bitleiste Gestoe_Slaves loeschen
      UC    "RDSYSST";
      {     P#L 50.0, P#L 16.0, P#L 0.0, P#L 14.0, P#L 50.1, P#L 51.0, P#L 57.0 };
      A     L 50.1;
      =     DIX 30.5;	//Ausgefallene Slaves
      BLD   8;	//-> werden zu Betr_Slaves
      AN    BR;	//-> werden zu Betr_Slaves_Mem
      ON    DIX 30.5;
      S     DIX 28.2;
      L     #RETVAL_SFC;
      L     W#16#8082;
      ==I;
      S     DIX 28.3;
RDCK: ON    DIX 28.0;
      ON    DIX 28.1;
      ON    DIX 28.2;
      JC    OUT;	//-> Anlauf Ende
//Gestoerte Slaves ermitteln aus Auswertung
//betroffene Slaves exclusiv mit ausgefallene Slaves.
//Die betroffenen Slaves werden zusaetzlich gespeichert.
      L     DID 1176;	//Slave ist betroffen =1
      L     DID 1192;	//-> sichern als Betr_Slave_Mem
      XOD;	//Slave ist ausgefallen =0
      T     DID 1208;
      L     DID 1180;	//-> Slave ist gestoert =1
      L     DID 1196;
      XOD;
      T     DID 1212;
      L     DID 1184;
      L     DID 1200;
      XOD;
      T     DID 1216;
      L     DID 1188;
      L     DID 1204;
      XOD;
      T     DID 1220;
      A     DIX 28.3;
      JCN   GEST;
      L     DW#16#0;
      T     DID 1224;
      T     DID 1228;
      T     DID 1232;	//Anlauf-/Resetbearbeitung fertig
      T     DID 1236;	//-> Datenausgabe
      L     DID 1208;
      T     DID 1240;
      T     DID 1256;
      L     DID 1212;
      T     DID 1244;
      T     DID 1260;
      L     DID 1216;
      T     DID 1248;
      T     DID 1264;
      L     DID 1220;
      T     DID 1252;
      T     DID 1268;
      JU    ANLE;
GEST: L     DID 1240;
      T     DID 1256;
      L     DID 1208;
      XOD;
      T     DID 1224;
      L     DID 1244;
      T     DID 1260;
      L     DID 1212;
      XOD;
      T     DID 1228;
      L     DID 1248;
      T     DID 1264;
      L     DID 1216;
      XOD;
      T     DID 1232;
      L     DID 1252;
      T     DID 1268;
      L     DID 1220;
      XOD;
      T     DID 1236;
ANLE: SET;
      S     DIX 28.4;
      JU    OUT;
NETWORK
TITLE = Verzweigung: Fehleranzahl ermitteln, Tippen (nur OB1)
//Zyklischer Betrieb: Dieser Teil wird immer im OB1 durchlaufen.
//Laeuft das Lesen der Diagnosedaten ueber SFC13, wird der SFC13 weiter 
//aufgerufen. Laeuft ein asnychroner SZL_C91-Leseauftrag, wird SZL C91 weiter
//gelesen. Liegen noch unbearbeitete Eintraege in der ULL, werden diese zuerst 
//abgearbeitet. Ansonsten wird die Anzahl der Betr_Slaves (betroffen = 
//ausgefallen oder gestoert) ermittelt. Sind keine betroffenen Slaves 
//(Betr_Slaves =0) vorhanden, wird das aktuelle Fach und das Diagnosefach 
//geloescht. Sind betroffene Slaves vorhanden, wird das Bit "ALL_DP_SLAVES_OK" 
//rueckgesetzt. Es wird unterschieden zwischen Automatik- und Handbetrieb 
//(Einzeldiagnose von Slaves). Im Automatikbetrieb wird bei Slave_Tippen bzw. 
//Fehler_Tippen in den Slave_Tipp-Betrieb bzw. Error_Tipp-Betrieb verzweigt. Wenn 
//bisher nicht getippt wurde, wird anschliessend geprueft, ob ein Slave bisher 
//betroffen war. Wenn ja, werden nur dann dessen neue Diagnosedaten gelesen, wenn 
//eine neue Diagnose des Slaves ansteht (OB82 / 86). Ansonsten wird das bisherige 
//aktuelle Fach ausgegeben. Im Handbetrieb wird die anparametrierte Slave-Nr. am 
//Parameter "SINGLE_DIAG_ADR" uebernommen und die Diagnose dieses Slaves gelesen. 
//In den Fehler-Tipp-Betrieb kann dann ebenfalls verzweigt werden.
AUSW: A     DIX 29.0;	//Solange SZL_C91-Lesen aktiv
      JC    C91;	//-> Weiter SZLC91-Lesen
      A     DIX 29.2;	//Wenn Folgeauftrag vorhanden
      JC    ULL;	//-> ULL bearbeiten
      LAR1  P##SZL_READ_C91;	//Startadresse C91-Fach (BGZD)
      L     DIB [AR1,P#0.0];	//Wenn Mastersystem-ID aus C91-Fach
      L     #MAST_SYSTEM_ID;	//nicht identisch mit Eingangsparameter
      <>I;
      =     DIX 30.4;	//-> Parametrierfehler
      JC    ENDE;	//-> Ende Baustein
      A     DIX 28.7;	//Solange SFC13-Lesen aktiv 
      JC    NMRD;	//-> Weiter SFC13-Lesen
//Anzahl Betroffene Slaves ermitteln
      L     0;	//Anzahl Betr_Slaves loeschen
      T     DIB 32;
      LAR1  P##AFFECT_SLAVES;	//Startadresse Bitleiste Betr_Slaves
      L     4;	//Anzahl DWorte in Bitleiste (4 DWORD)
NXW1: T     #LOOP_CNT_2;	//-> Schleifenzaehler aussen
      L     DID [AR1,P#0.0];	//Aktuelles Wort der Bitleiste sichern
      T     #TEMP_VAR_1;	//als Zwischenwert sichern
      L     32;	//Anzahl der Bits im DWort (32 Bits)
NXB1: T     #LOOP_CNT_1;	//-> Schleifenzaehler innen
      L     #TEMP_VAR_1;	//Unterstes Bit rausschieben
      SLD   1;
      T     #TEMP_VAR_1;	//und als neuen Wert wieder sichern
      JZ    CON1;
      L     DIB 32;	//Wenn Bit gesetzt
      INC   1;	//-> Summe inkrementieren 
      T     DIB 32;
CON1: L     #LOOP_CNT_1;	//Naechstes Bit im DWort pruefen
      LOOP  NXB1;
      +AR1  P#4.0;	//Naechstes DWort der Bitleiste pruefen
      L     #LOOP_CNT_2;
      LOOP  NXW1;
      L     DIB 32;	//Wenn Anzahl Betr_Slaves <>0
      L     0;
      <>I;
      R     DIX 4.0;	//-> Alles_O.K.-Bit ruecksetzen
//Unterscheidung Hand- und Automatikbetrieb
      LAR1  DID 34;	//Slave_Tippindex = Angezeigter Slaves
      AN    DIX 1402.1;
      JC    AUTO;
//Betriebsart: Hand
      R     DIX 30.2;	//Slave_Suchen-Start ruecksetzen
      L     P##AFFECT_SLAVES;	//Startadr. Bitfeld betr. Slaves 
      T     DID 34;	//-> Slave_Tippindex
      L     DIB 1403;	//Angegebene Slave_Nr. sichern
      T     DIW 50;
// 
      A     DIX 1402.5;	//Wenn Einzeldiagnose aktiviert
      FP    DIX 29.6;
      =     DIX 29.1;
      JC    DIAN;	//-> Diagnose lesen
      LAR2  P##ACT_DAT;	//Startadresse aktuelles Fach
      A     DIX [AR2,P#1.0];	//Wenn angegebener Slave 
      X     DIX [AR2,P#1.1];	//ausgefallen oder gestoert
      A     DIX 1402.3;	//und Error_Tippen aktiviert
      FP    DIX 29.4;
      JC    T_ER;	//-> Error_Tipp-Betrieb bearbeiten
      JU    OUT;	//sonst weiter Datenausgabe
//Betriebsart: Automatik
AUTO: A     DIX 4.0;	//Wenn keine Slaves betroffen
      JC    OK;	//-> Loeschen des akt. Faches 
//Es sind betroffene Slaves vorhanden
      A     DIX 1402.2;	//Wenn Slave_Tippen aktiviert
      FP    DIX 29.3;
      JC    T_SL;	//-> Slave_Tipp-Betrieb bearbeiten
// 
      A     DIX [AR1,P#0.0];	//Wenn angezeigter Slave noch betroffen
      A     DIX 1402.3;	//und Error_Tippen aktiviert
      FP    DIX 29.4;
      JC    T_ER;	//-> Error_Tipp-Betrieb bearbeiten
      A     DIX 29.7;	//Wenn Slave_Tipp-Betrieb aktiv
      A     DIX [AR1,P#0.0];	//und angezeigter Slave noch betroffen
      A     DIX 28.5;	//und neue Diagnose
      JC    DIAG;	//-> Diagnose auswerten
      A     DIX 29.7;	//Wenn Slave_Tipp-Betrieb aktiv
      A     DIX [AR1,P#0.0];	//und angezeigter Slave noch betroffen
      AN    DIX 28.5;	//aber keine neue Diagnose
      JC    OUT;	//-> weiter Datenausgabe
      A     DIX 30.2;	//Wenn Slave_Such-Betrieb aktiv
      A     DIX [AR1,P#0.0];	//und angezeigter Slave noch betroffen
      A     DIX 28.5;	//und neue Diagnose
      JC    DIAG;	//-> Diagnose auswerten
      A     DIX 30.2;	//Wenn Slave_Such-Betrieb aktiv
      A     DIX [AR1,P#0.0];	//und angezeigter Slave noch betroffen
      AN    DIX 28.5;	//aber keine neue Diagnose
      JC    OUT;	//-> weiter Datenausgabe
      JU    FRST;	//sonst ersten Betr_Slave suchen
//Es sind keine betroffenen Slaves vorhanden 
OK:   LAR2  P##ACT_DAT;	//Aktuelles Fach loeschen
      L     DW#16#0;
      T     DID [AR2,P#0.0];
      T     DID [AR2,P#4.0];
      T     DID [AR2,P#8.0];
      T     DID [AR2,P#12.0];
      T     DID [AR2,P#16.0];
      T     DIW [AR2,P#20.0];
      LAR1  P##DIAG_DAT_NORM;	//Diagnosefach loeschen
      L     61;	//Anzahl: 244 Bytes = 61 Dword
BEGN: T     #LOOP_CNT_1;	//-> Schleifenzaehler
      L     DW#16#0;
      T     DID [AR1,P#0.0];	//Dword loeschen
      +AR1  P#4.0;	//naechstes Dword
      L     #LOOP_CNT_1;
      LOOP  BEGN;
      JU    OUT;	//-> Datenausgabe
NETWORK
TITLE = Ersten betroffenen Slave ermitteln
//Aus der Bitleiste der Betr_Slaves wird die erste betroffene Slave-Nr. 
//ermittelt. Wird ird kein Slave gefunden, erfolgt als Loeschen "Summe betroffene 
//Slaves". 
FRST: A     DIX 30.2;	//Wenn erstmaliges Slave-Suchen
      JC    NSRH;
      S     DIX 30.2;	//-> Slave_Suchen-Start setzen
NSRH: LAR1  P##AFFECT_SLAVES;	//Startadresse Bitleiste Betr_Slaves
      L     4;	//Anzahl DWorte in Bitleiste (4 DWORD)
NXW2: T     #LOOP_CNT_2;	//-> Schleifenzaehler aussen
      L     DID [AR1,P#0.0];	//Aktuelles Wort der Bitleiste
      CAD;	//ausrichten (Bytes tauschen)
      T     #TEMP_VAR_1;	//als Zwischenwert sichern
      L     32;	//Anzahl der Bits im DWort (32 Bits)
NXB2: T     #LOOP_CNT_1;	//-> Schleifenzaehler innen
      L     #TEMP_VAR_1;	//Unterstes Bit rausschieben
      SRD   1;
      T     #TEMP_VAR_1;	//und als neuen Wert wieder sichern
      JN    GEF;	//Wenn Bit gesetzt -> Slave_Nr. sichern 
      L     #LOOP_CNT_1;	//Naechstes Bit im DWort pruefen
      LOOP  NXB2;
      +AR1  P#4.0;	//Naechstes DWort der Bitleiste pruefen
      L     #LOOP_CNT_2;
      LOOP  NXW2;
      L     0;	//Wenn kein Slave gefunden 
      T     DIB 32;	//-> Anzahl Betr_Slaves =0
      JU    ENDE;	//-> Ende Baustein
GEF:  L     4;	//Slave_Nr. berechnen aus
      L     #LOOP_CNT_2;	//(Anz.DWorte - SCHLEIFE_2) * 32
      -I;	//+ (Anz.Bits - SCHLEIFE_1 + 1)
      L     32;
      *I;
      T     #TEMP_VAR_1;
      L     32;
      L     #LOOP_CNT_1;
      -I;
      INC   1;
      L     #TEMP_VAR_1;
      +I;
      T     DIW 50;	//-> Slave_Nr.
      L     8;	//:8 -> Akku1-L (Byteadresse) 
      /I;
      T     #TEMP_VAR_1;	//   -> Akku1-H (Bitadresse)
      AD    DW#16#FFFF;
      T     #TEMP_VAR_2;	//Byte-Nr. sichern
      L     DW#16#0;
      L     #TEMP_VAR_1;
      SRD   16;	//Bitadresse ermitteln
      <>D;	//Wenn Bitadresse <>0
      JC    GAN4;	//-> Bitadresse sofort dekrementieren
      L     B#16#8;	//sonst Bitadr.=8 -> spaeter dekrement.
      T     #TEMP_VAR_1;	//sichern
      L     #TEMP_VAR_2;
      DEC   1;	//Byte-Nr. dekrementieren
      T     #TEMP_VAR_2;
      TAK;
GAN4: DEC   1;	//Bitadresse dekrementieren
      L     #TEMP_VAR_2;
      SLD   3;	//Gesamtadresse = Byteadresse
      +D;	//+ Bitadresse
      L     P##AFFECT_SLAVES;	//+ Startadresse Betr_Slaves
      +D;
      T     DID 34;	//-> neuer Tippindex
      JU    DIAN;	//-> Diagnosedaten neu lesen
NETWORK
TITLE = Tippen der Diag Slaves (Slave_Tippen)
//Wenn Slave_Tipp-Betrieb eingeschaltet, wird ueber Tippen (Flanke) der naechste 
//betroffene Slave in der Bitleiste Betr_Slaves gesucht (Durchwahl der Slaves). 
//Die Suche nach neuen Slaves startet ab der aktuell angezeigten Slave-Nr. 
//(Slave-Tippindex). Wird ein neuer Slave gefunden, wird der Tippindex auf die 
//neue betroffene Slave-Nr. gesetzt. Sind alle Fehler durchgetippt, wird wieder 
//bei der ersten betroffenen Slave-Nr. begonnen.
//Beachte: Erster Slave beginnt bei Adresse 0.0
T_SL: A     DIX 29.7;	//Wenn erstmaliges Slave_Tippen
      JC    NXTP;
      S     DIX 29.7;	//-> Slave_TIPP-Start setzen
NXTP: LAR1  DID 34;	//Aktueller Slave_Tippindex
      L     P#0.1;	//+ 1
      +AR1;	//-> Adresse des "naechsten" Slaves
      L     DIW 50;	//-> Slave_Nr.          
      INC   1;
      T     DIW 50;
      L     P##AFFECT_SLAVES;	//Adresse Slave_1
      L     P#15.5;	//+ Offset Slave_126
      +D;
      T     #TEMP_VAR_1;	//-> Adresse des "letzten" Slaves
      L     126;	//Schleifenzaehler = max. Slaveanzahl
LOP7: T     #LOOP_CNT_1;
      TAR1;	//Adresse des aktuellen Slaves
      L     #TEMP_VAR_1;	//Adresse des letzten Slaves
      <=I;	//Wenn Adresse gueltig
      JC    NSLV;	//-> Naechsten Slave pruefen
      LAR1  P##AFFECT_SLAVES;	//sonst wieder bei Slave_1 starten
      L     1;	//Slave_Nr. = Slave_1
      T     DIW 50;
NSLV: A     DIX [AR1,P#0.0];	//Wenn Slave betroffen
      JC    NGEF;	//-> Gefundenen Slave auswerten
      L     DIW 50;
      INC   1;	//sonst erhoehen Slave_Nr.
      T     DIW 50;
      +AR1  P#0.1;	//naechsten Slave pruefen
      L     #LOOP_CNT_1;
      LOOP  LOP7;
NGEF: TAR1  DID 34;	//Neuer Tippindex = neue Slave_Nr.
      JU    DIAN;	//-> Diagnosedaten neu lesen
NETWORK
TITLE = Slave_Nr. wandeln in Diagnoseadresse, Diagnosedaten lesen
//Vorab wird das aktuelle Fach initialisiert. Mit dem SFC5 wird die aktuelle 
//geographische Slave-Adresse in eine Diagnoseadresse gewandelt, die in das
//aktuelle Fach eingetragen wird. Danach werden die Diagnosedaten des Slaves mit
//SFC13 gelesen und ausgewertet. Der nicht beschriebene Bereich des Diagnose- 
//faches wird geloescht. Am SFC13 wird die vorher ermittelte Diagnoseadresse 
//anparametriert. Der Slave-Stellvertreter ist beim alten S7-Slotmodell immer der 
//Steckplatz 2 (sowohl bei modularen als auch bei kompakten DP-Slaves). Beim 
//neuen DPV1-Slotmodell hat der Slave-Stellvertreter den Steckplatz 0. 
//Die Diagnoseinfos werden aus dem Diagnosefach in das aktuelle Fach kopiert. 
//Bei einem gestoerten o. ausgefallenen Slave wird sofort danach der erste Fehler 
//ausgewertet. Wenn im Fehler-Tipp-Betrieb waehrend der Fehleranzeige eines 
//betroffenen Slaves ein neues Ereignis (OB82/OB86) eintritt, wird nur dann die 
//Diagnose neu gelesen, wenn das Ereignis zum dem aktuell angezeigten Slaves 
//passt. Bei Hand-Einzeldiagnose wird die Diagnose immer gelesen und ausgwertet.
DIAG: R     DIX 28.5;	//Diagnose wird bearbeitet
      AN    DIX 28.6;	//Wenn Diagnose nicht zum Slave passt
      JC    OUT;	//-> weiter Datenausgabe
DIAN: R     DIX 28.5;	//Neue Diagnose wird bearbeitet
      R     DIX 28.6;
      LAR2  P##ACT_DAT;	//Startadresse aktuelles Fach
      L     DW#16#0;	//Aktuelles Fach loeschen 
      T     DID [AR2,P#0.0];
      T     DID [AR2,P#4.0];
      T     DID [AR2,P#8.0];
      T     DID [AR2,P#12.0];
      T     DID [AR2,P#16.0];
      T     DIW [AR2,P#20.0];
      L     DIW 50;	//Slave_Nr.
      T     DIB [AR2,P#0.0];	//in akt. Fach eintragen
//Geographische Slave_Adresse in logische Slave_Adresse wandeln
//Erster Versuch mit Slave-Stellvertreter 黚er Slot =0 (DPV1-Modell)
//Zweiter Versuch mit Slave-Stellvertreter 黚er Slot =2 (S7-Modell)
      L     W#16#0;	//Slot des Slave-Stellvertreters
NOV1: T     #SLOT_SFC49_5;
      CALL  "GADR_LGC" (
           SUBNETID                 := #SUBNET_ID,
           RACK                     := DIW 50,
           SLOT                     := #SLOT_SFC49_5,
           SUBSLOT                  := B#16#0,
           SUBADDR                  := W#16#0,
           RET_VAL                  := #RETVAL_SFC,
           IOID                     := #IO_FLAG,
           LADDR                    := #DIAG_ADDR);	//Slave geografisch -> logisch / Mastersystem-ID / Slave_Nr. / Slot des Slave-Stellvertreters / Diagnoseadresse temp. sichern
      AN    BR;	//Wenn Fehler bei SFC5-Bearbeitung
      A     DIX 31.4;	//und beide Slot-Modelle geprueft 
      R     DIX 31.4;
      JC    ERDG;	//-> Fehlerroutine
      AN    BR;	//Wenn Fehler bei SFC5-Bearbeitung
      =     DIX 31.4;	//-> kein DPV1-Slot-Modell
      L     W#16#2;	//-> S7-Slot-Modell pruefen
      JC    NOV1;	//-> neuer SFC5-Aufruf
      L     #DIAG_ADDR;	//Diagnoseadresse
      T     DIW [AR2,P#6.0];	//in akt. Fach eintragen
//DP-Normdiagnose des betroffenen Slaves (weiter) lesen
NMRD: LAR2  P##ACT_DAT;	//Startadresse aktuelles Fach
      L     DIW [AR2,P#6.0];	//Diagnoseadresse
      T     #DIAG_ADDR;	//temp. sichern
      BLD   7;	//Norm-Diagnosedaten lesen
      SET;
      =     L 50.0;	//Diagnoseadresse
      L     W#16#1002;
      T     LW 51;	//Datenfach fuer SFC13-Daten
      L     244;
      T     LW 53;	//Laenge SFC13-Daten sichern
      L     DINO;
      T     LW 55;	//Wenn Fehler bei SFC13-Bearbeitung
      L     P#DBX 932.0;	//-> SFC13_Lesen deaktivieren
      T     LD 57;	//-> Fehlerroutine
      UC    "DPNRM_DG";	//Wenn SFC13-Lesen beendet
      {     P#L 50.0, P#L 24.0, P#L 14.0, P#L 51.0, P#L 50.1 };	//-> SFC13_Lesen deaktivieren
      A     L 50.1;	//-> Diagnosedaten auswerten
      =     DIX 30.5;	//sonst SFC13_Lesen aktivieren
      BLD   8;	//-> Ende Baustein
//Diagnosedaten auswerten und in Aktuelles Fach eintragen
      L     #RETVAL_SFC;	//Startadresse Diagnosefach
      T     DIB 44;	//Wenn "Diag_Ext_Diag"
      AN    BR;	//oder "Diag_State_Diag"
      R     DIX 28.7;	//-> Status: Slave_gestoert
      JC    ERDG;	//Wenn "Station_Non_Exist"
      AN    DIX 30.5;	//oder "Station_Not_Ready"
      R     DIX 28.7;	//oder "Invalid_Slave_Response" 
      JC    DAUS;	//oder "Diag_Prm_Request"
      S     DIX 28.7;	//oder "Diag_Deactivated"
      JU    ENDE;	//-> Status: Slave_ausgefallen
DAUS: LAR1  P##DIAG_DAT_NORM;	//-> Status: Slave_gestoert reset
      A     DIX [AR1,P#0.3];	//PNO-ID des DP-Slaves
      O     DIX [AR1,P#1.1];	//in akt. Fach eintragen
      S     DIX [AR2,P#1.1];	//-> Restliche Diagnosedaten loeschen
//Fehlerroutine bei SFC13- oder SFC5-Bearbeitung
      A     DIX [AR1,P#0.0];	//Startadresse Diagnosefach
      O     DIX [AR1,P#0.1];
      O     DIX [AR1,P#0.5];	//-> Status: Slave_nicht_projektiert
      O     DIX [AR1,P#1.0];
      O     DIX [AR1,P#1.7];	//Diagnoselaenge =0 setzen
//Restlicher nicht beschriebener Bereich im Diagnosefach loeschen
      S     DIX [AR2,P#1.0];	//Startadresse Diagnosefach
      R     DIX [AR2,P#1.1];	//+ Offset Diagnoselaenge_SFC13
      L     DIW [AR1,P#4.0];	//-> Startadresse Restdaten
      T     DIW [AR2,P#2.0];	//Gesamtlaenge Diagnosefach
      JU    DLDG;	//- Aktuelle Laenge Slavediagnose
ERDG: LAR1  P##DIAG_DAT_NORM;
      L     B#16#3;	//-> Schleifenzaehler
      T     DIB [AR2,P#1.0];	//Byte loeschen
      L     B#16#0;
      T     DIB 44;	//naechstes Byte
DLDG: L     DIB 44;
      SLD   3;
//Slave-Diagnosedaten gelesen: Error-Tippen initialisieren. 
//Auto: Wenn Slave gestoert o. ausgefallen, Uebergang in Error-Tipp-Betrieb 
//Hand: Wenn Slave-Einzeldiagnose aktiv, Uebergang in Error-Tipp-Betrieb
      +AR1;	//Akt. Diaglaenge initialisieren
      L     244;	//mit 6 Bytes Normdiagnose
      L     DIB 44;
      -I;	//Fehlernummer =0
DEL:  T     #LOOP_CNT_1;	//Laenge Diagnoseblock =0
      L     B#16#0;
      T     DIB [AR1,P#0.0];	//Error_Tippindex =Start Diagnose
      +AR1  P#1.0;
      L     #LOOP_CNT_1;	//Grundzustand Error_Tippen
      LOOP  DEL;	//Grundzustand Blockauswertung
      L     6;	//Kennungsdiagnose initialisieren
      T     DIB 45;	//Kanaldiagnose initialisieren
      L     0;	//S7-Diagnosealarm initialisieren
      T     DIB 49;	//S7-Diagnose initialisieren
      T     DIB 46;	//Wenn Einzeldiagnose aktiviert
      L     P##DIAG_DAT_NORM;	//-> sofort Diagnose auswerten
      T     DID 38;	//Wenn Slave ausgefallen o. gestoert
      SET;	//-> sofort Diagnose auswerten
      R     DIX 30.0;	//sonst Datenausgabe
      R     DIX 30.1;
      R     DIX 30.7;
      R     DIX 31.0;
      R     DIX 31.1;
      R     DIX 31.2;
      A     DIX 29.1;
      JC    T_ER;
      A     DIX [AR2,P#1.0];
      X     DIX [AR2,P#1.1];
      JCN   OUT;
NETWORK
TITLE = Tippen der Fehler pro Slave (Error_Tippen)
//Wenn Error_Tipp-Betrieb eingeschaltet, wird ueber Tippen (Flanke) der naechste 
//Fehler im Diagnosetelegramm des betroffenen Slave gesucht (Durchwahl der 
//Fehler). Die Suche nach dem neuen Fehler startet ab der aktuell angezeigten 
//Fehler-Nr. (Error-Tippindex). Wird ein neuer Fehler gefunden, wird der 
//Tippindex auf den neuen Fehler gesetzt.
//Ueber einen Sprungverteiler wird unterschieden zwischen Kennungsdiagnose, 
//Modulstatus, Kanaldiagnose DS0/DS1-Diagnose (S7-Slave) und hersteller- 
//spezifische Geraetediagnose. Der Fehlertyp wird durch den Parameter ERROR_TYP 
//beschrieben, ueber die ERROR_NR werden die einzelnen Fehler voneinander 
//unterschieden. Sind alle Fehler durchgetippt, wird wieder bei dem Fehler mit 
//der Nr.1 begonnen. Das Fehlertippen wird zurueckgesetzt, wenn ein Slave-Tippen 
//erfolgt, d.h. Slave-Tippen hat eine hoehere Prioritaet als Error-Tippen.
//Jedem Kanal-Fehler wird ein eindeutiger Fehler-Code zugeordnet und in 
//"CHANNEL_ERROR_CODE" abgelegt. Zusaetzlich werden aller Fehler bitcodiert in 
//CHANNEL_ERROR_INFO eingetragen.
//Besteht die Gesamtdiagnose neben der Kennungsdiagnose aus weiteren Diagnose-
//bloecken (z.B. Kanal- und/oder Geraetediagnose), dann wir die Auswertung der 
//Kennunsgdiagnose uebersprungen (wenig Aussagekraft). Wenn bei S7-Slaves aber
//erkannt wird, da� in der Alarminfo (DS0/1) keine Details stehen, erfolgt 
//anschliessend die Auswertung der anfaenglich uebersprungenen Kennungsdiagnose 
//(besser wenig Infos als keine Infos).   
T_ER: A     DIX 30.0;	//Wenn erstmaliges Error_Tippen
      JC    NXER;
      S     DIX 30.0;	//-> Error_TIPP-Start setzen
      JC    NBLK;	//-> Neuer Diagnoseblock auswerten
NXER: L     P##DIAG_DAT_NORM;	//Startadresse Diagnosefach
      L     DIB 45;	//+ Aktuelle Gesamtdiagnoselaenge
      SLD   3;
      +D;	//-> Endadresse akt. Diagnoseblock
      L     DID 38;	//> Error_Tippindex
      >I;
      JC    GBLK;	//-> Weiterhin im gleichen Block
//Neuen Diagnoseblock auswerten
NBLK: R     DIX 30.1;	//Start Diagnoseblock ruecksetzen   
      LAR1  P##DIAG_DAT_NORM;	//Startadresse Diagnosefach
      L     DIB 45;	//+ Aktuelle Gesamtdiagnoselaenge
      SLD   3;
      +AR1;	//-> Startadr. neuer Diagnoseblock
      TAR1  DID 52;	//Startadresse sichern
      TAR1  DID 38;	//Tippindex = Startadr. Diagblock 
      L     DIB [AR1,P#0.0];	//Headerkennung des Diagnoseblocks
      SRW   6;
      T     DIB 47;	//sichern
      L     B#16#3;	//Wenn Kennung fuer Revision 
      <>I;
      JC    NDIA;
//Auswertung Revision (immer 1 Byte lang)
      L     DIB 45;	//-> Aktuelle Gesamtdiagnoselaenge +1
      INC   1;
      T     DIB 45;
      JU    BEND;	//-> Ende Diagnoseblock
//Ueberpruefung der Laenge des Diagnosebloecks 
NDIA: L     DIB [AR1,P#0.0];	//Akt. Header (Kennung ausmaskieren)
      AW    W#16#80;	//Wenn kanalbezogene Diagnose erkannt
      L     B#16#3;	//3 Byte Laenge Kanaldiagnose (fest)        
      JN    KANL;	//-> temp. sichern
      L     DIB [AR1,P#0.0];	//Akt. Header (Kennung ausmaskieren)
      AW    W#16#3F;	//-> Laenge des Diagnoseblocks
KANL: T     DIB 46;	//temp. sichern
      L     DIB 45;	//+ aktuelle Gesamtdiagnoselaenge
      +I;
      T     DIB 45;	//-> neue akt. Gesamtdiagnoselaenge
      L     DIB 44;	//Laenge Diag.Block + akt.Gesamtlaenge
      >I;	//> als SFC13-Diagnoselaenge
      JC    OUT;	//-> keine weitere Auswertung
      L     DIB 46;	//Wenn Laenge des Diagnoseblocks =0
      L     B#16#0;
      ==I;
      JC    OUT;	//-> Datenausgabe
//Auswertung der Diagnosebloecke
GBLK: L     DIB 47;	//Headerkennung der Diagnose
      JL    KUNG;	//Wenn Kennung ungueltig -> Ende Auswertung
      JU    GERB;	//-> Auswertung Geraetebez. Diagnose(00)
      JU    KENB;	//-> Auswertung Kennungsbez. Diagnose(01)
      JU    KANB;	//-> Auswertung Kanalbez. Diagnose(10)
KUNG: JU    KAUS;	//ungueltig -> keine Auswertung
//Beginn Auswertung Geraetebezogene Diagnose
//Es wird unterschieden zwischen Modulstatus, Leitungsdiagnose,
//DS0/1 bei S7-Slaves und herstellerspezifischen Diagnoseinfos.
GERB: LAR1  DID 52;	//Startadresse DiagBlock
      LAR2  P##ACT_DAT;	//Startadresse aktuelles Fach 
      A(;
      L     DIB [AR1,P#1.0];	//Wenn Modulstatus erkannt
      L     B#16#82;	//Byte 1-3: 82 00 00
      ==I;
      );
      A(;
      L     DIW [AR1,P#2.0];
      L     0;
      ==I;
      );
      JC    MLGO;	//-> Modulstatus-Auswertung
//Wenn PNO-ID =80xx -> Siemens-Slave 
      L     DIW [AR2,P#2.0];	//Wenn PNO_ID des Slaves <>80xx
      SRW   8;
      L     W#16#80;
      <>I;
      =     DIX 31.3;	//-> keine Diagnoseinfos vorhanden
      JC    KAUS;	//-> allg. Geraetediganose
//Pruefe, ob Siemens-Leitungsdiagnose vorliegt
      L     DIB 46;	//Wenn Laenge Diagnoseblock <>19
      L     B#16#13;	//-> keine Leitungsdiagnose
      <>I;
      JC    CKS7;
      L     DIB [AR1,P#1.0];	//Wenn keine Leitungsdiagnose erkannt
      L     B#16#A0;
      <>I;
      JC    CKS7;	//-> Pruefe, ob S7-Slave
//Leitungsdiagnose erkannt:
      L     DW#16#0;	//Initialisieren: Steckplatznummer,
      T     DID [AR2,P#8.0];	//Modulstatus, Kanalnummer, Kanaltyp
      T     DID [AR2,P#12.0];	//Kanal-Fehlerinfos_1
      T     DID [AR2,P#16.0];	//Kanal-Fehlerinfos_2
      T     DIW [AR2,P#20.0];	//Error-Code
      L     DIB [AR1,P#6.0];	//Wenn Fehlerrate =FFh
      L     B#16#FF;	//-> keine Störung im Segment
      ==I;
      JC    BEND;	//-> Ende Diagnoseblock
//Stoerung im Segment 
      L     B#16#6;	//Error_Typ =6 
      T     #SUM_SLAVES_DIAG;	//in akt. Fach eintragen
      L     DIB 49;	//Fehlernummer inkrementieren
      INC   1;
      T     DIB 49;
      T     DIB [AR2,P#4.0];	//und in akt. Fach eintragen
      L     DIB [AR1,P#4.0];	//sonst Segmentnummer ermitteln
      SRW   4;
      JL    SGER;
      JU    SGER;
      JU    SG03;	//Segment 3
      JU    SG02;	//Segment 2
      JU    SGER;
      JU    SG01;	//Segment 1
      JU    SGER;
      JU    SGER;
      JU    SGER;
      JU    SG04;	//Segment 4
SGER: L     0;
      JU    SGMT;
SG03: L     3;
      JU    SGMT;
SG02: L     2;
      JU    SGMT;
SG01: L     1;
      JU    SGMT;
SG04: L     4;	//Segmentnummer
SGMT: T     #ERROR_NO;	//in akt. Fach eintragen
      L     DIB [AR1,P#6.0];	//Fehlerrate
      T     #ERROR_TYPE;	//in akt. Fach eintragen
      L     B#16#7F;
      L     DIB [AR1,P#7.0];	//Station x lesen
      AW    W#16#7F;	//Wenn Station x =7F
      <>I;	//-> Station x =FF setzen
      JC    STAX;
      L     B#16#FF;
STAX: T     #MODULE_NO;	//Station x in akt. Fach eintragen
      L     B#16#7F;
      L     DIB [AR1,P#8.0];	//Station y lesen
      AW    W#16#7F;	//Wenn Station y =7F
      <>I;	//-> Station y =FF setzen
      JC    STAY;
      L     B#16#FF;
STAY: T     #MODULE_STATE;	//Station y in akt. Fach eintragen
      A     DIX [AR2,P#12.7];	//Wenn ungueltige Station x
      L     W#16#FFFF;	//-> Entfernung von x =FFFF setzen
      JC    EFGX;
      L     DIW [AR1,P#9.0];	//Entfernung von x
      L     10;	//in Meter umrechnen
      /I;
EFGX: T     DIW [AR2,P#14.0];	//Entf. von x in akt. Fach eintragen
      A     DIX [AR2,P#13.7];	//Wenn ungueltige Station y
      L     W#16#FFFF;	//-> Entfernung von y =FFFF setzen
      JC    EFGY;
      L     DIW [AR1,P#11.0];	//Entfernung von y
      L     10;	//in Meter umrechnen
      /I;
EFGY: T     #CHANNEL_ERROR_CODE;	//Entf. von y in akt. Fach eintragen
      L     DIW [AR1,P#13.0];	//Entfernung von DR
      L     10;	//in Meter umrechnen
      /I;
      T     DIW [AR2,P#18.0];	//Entf. von DR in akt. Fach eintragen
      L     DID [AR1,P#15.0];	//Fehlerursache 
      CAD;	//Tausche Akku-Inhalte (LL,LH,HL,HH)
      T     #TEMP_VAR_1;	//-> sichern
      L     545;	//Error-Code initialisieren
      T     #TEMP_VAR_2;	//-> sichern
//Ermittlung der Bits in der Fehlerursache -> Bildung eindeutiger Error-Code
      L     32;	//Anzahl der Bits im Dword (32)
NXB5: T     #LOOP_CNT_1;	//-> Schleifenzaehler
      L     #TEMP_VAR_2;
      INC   1;	//Error_Code erhoehen
      T     #TEMP_VAR_2;
      L     #TEMP_VAR_1;	//Unterstes Bit rausschieben
      SRD   1;
      T     #TEMP_VAR_1;	//Wenn Fehlerbit gesetzt
      JN    ERUS;	//-> Error_Code generieren
      L     #LOOP_CNT_1;
      LOOP  NXB5;
ERUS: L     #TEMP_VAR_2;	//Error_Code
      T     DIW [AR2,P#20.0];	//in akt. Fach eintragen 
      L     DID 38;	//Error_Tippindex inkrementieren
      L     DIB 46;	//um die Laenge des Diagnoseblocks
      SLD   3;
      +D;
      T     DID 38;
      L     P##DIAG_DAT_NORM;	//Gesamtlaenge der Diagnose 
      L     DIB 44;
      SLD   3;
      +D;
      L     DID 38;	//> Error_Tippindex
      >D;
      JC    OUT;	//-> Datenausgabe 
      JU    DEND;	//sonst Diagnoseende erreicht
//Pruefe, ob S7-Slave vorliegt (8 <= Blocklaenge <= 48)
CKS7: L     DIB 46;
      L     B#16#30;	//Wenn Laenge Diagnoseblock >48 (DS1)
      >I;
      =     DIX 31.3;	//-> keine Diagnoseinfos vorhanden
      JC    KAUS;	//-> kein DS1 -> allg. Geaetediagnose
      TAK;
      L     B#16#8;	//Wenn Laenge Diagnoseblock <8 (DS0)
      <I;
      =     DIX 31.3;	//-> keine Diagnoseinfos vorhanden
      JC    KAUS;	//-> kein DS0 -> allg. Geaetediagnose
//S7-Slave erkannt: 
//Pruefen, ob Diagnosealarm und S7-Baugruppenstoerung vorhanden
      A     DIX 30.1;	//Wenn erstmalige Blockauswertung
      JC    DSGO;
      S     DIX 30.1;	//-> Start Diagnoseblock setzen
      LAR1  DID 52;	//Startadresse Diagblock
      L     DIB [AR1,P#1.0];	//Wenn kein Diagnosealarm (komm/geh) 
      L     B#16#1;
      <>I;
      =     DIX 31.3;	//-> keine Diagnoseinfos vorhanden
      JC    KAUS;	//-> Keine weitere Auswertung 
      S     DIX 31.1;	//sonst S7-Diagnosealarm vorhanden
      AN    DIX [AR1,P#4.0];	//Wenn gehender S7-Diagnosealarm 
      JC    KAUS;	//-> Keine weitere Auswertung 
      S     DIX 31.2;	//sonst kommende S7-Diagnose (DS0/1)
//DS0/1 liegt vor:
      L     DW#16#0;	//Initialisieren: Steckplatznummer,
      T     DID [AR2,P#8.0];	//Modulstatus, Kanalnummer, Kanaltyp
      T     DID [AR2,P#12.0];	//Kanal-Fehlerinfos_1
      T     DID [AR2,P#16.0];	//Kanal-Fehlerinfos_2
      T     DIW [AR2,P#20.0];	//Error-Code
      L     B#16#4;	//Error_Typ =4 
      T     #SUM_SLAVES_DIAG;	//in akt. Fach eintragen
      L     DIB [AR1,P#2.0];	//Steckplatznummer
      T     DIB [AR2,P#8.0];	//in akt. Fach eintragen
//Die ersten 4 Bits und die Baugruppenklasse werden nicht beruecksichtigt
      L     DID [AR1,P#4.0];	//DS0 als Kanal-Fehlerinfos_2 
      T     DID [AR2,P#16.0];	//in akt. Fach eintragen
      CAD;	//Tausche Akku-Inhalte (LL,LH,HL,HH)
      AD    DW#16#FFFF00F0;	//Fehlerinfos ausmaskieren
      T     #TEMP_VAR_1;	//-> sichern
      L     512;	//Error-Code initialisieren
      T     #TEMP_VAR_2;	//-> sichern
//Ermittlung der Bits in der Fehlerinfo -> Bildung eindeutiger Error-Code
      L     32;	//Anzahl der Bits im Dword (32)
NXB3: T     #LOOP_CNT_1;	//-> Schleifenzaehler
      L     #TEMP_VAR_2;
      INC   1;	//Error_Code erhoehen
      T     #TEMP_VAR_2;
      L     #TEMP_VAR_1;	//Unterstes Bit rausschieben
      SRD   1;
      T     #TEMP_VAR_1;
      JN    ERIF;
      L     #LOOP_CNT_1;
      LOOP  NXB3;
ERIF: L     #TEMP_VAR_2;	//Error_Code
      T     DIW [AR2,P#20.0];	//in akt. Fach eintragen 
      L     DIB 46;	//Wenn Laenge Diagnoseblock =8 (DS0)
      L     B#16#8;
      ==I;
      JC    NCHL;	//-> keine DS1-Auswertung
//Pruefen, ob Bitgranulare Peripherie (z.B. ASI-CP) vorhanden
      L     DIB [AR1,P#8.0];	//Kanaltyp (nach S7)
      T     #ERROR_TYPE;	//in akt. Fach eintragen
      L     W#16#60;	//Wenn Kanaltyp
      <>I;	//bitgranulare Peripherie
      JC    NBIT;
      L     32;	//Error_Code =32
      T     DIW [AR2,P#20.0];	//in akt. Fach eintragen
      L     DID [AR1,P#11.0];	//Bitfeld Teil_1
      T     DID [AR2,P#12.0];	//in akt. Fach eintragen
      L     DIB [AR1,P#10.0];	//Wenn Anzahl gleichart. Kanaele >32
      L     W#16#20;
      <=I;
      JC    NBIT;
      L     DID [AR1,P#15.0];	//-> Bitfeld Teil_2
      T     DID [AR2,P#16.0];	//in akt. Fach eintragen
//Pruefen, ob Kanalfehler vorhanden
NBIT: L     DIB [AR1,P#8.0];	//Kanaltyp (nach S7)
      SRW   4;
      L     W#16#7;	//Wenn Kanaltyp 
      <>I;	//ohne Kanalinformationen
      JC    NCHL;	//-> keine Kanalauswertung
      L     DIB [AR1,P#9.0];	//Wenn Anzahl Diagnosebits pro Kanal =0
      L     B#16#0;
      ==I;
      JC    NCHL;	//-> keine Kanalauswertung
      L     DIB [AR1,P#11.0];	//Wenn Anzahl Kanalfehler =0
      ==I;
      JC    NCHL;	//-> keine Kanalauswertung
      L     -1;	//Initialisieren
      T     #ERROR_NO;	//Kanalnummer (Start mit Kanal 0)
      L     DIB [AR1,P#10.0];	//Anzahl der gleichartigen Kanaele
      T     DIB 48;	//-> Indexzaehler im Diagnoseblock
      L     DID 52;	//Startadresse Diagblock
      L     P#11.0;	//+ Kopf und Offset im DS1
      +D;
      T     DID 38;	//-> neuer Tippindex
      LAR1;
DSGO: L     DIB 48;	//Indexzaehler im Diagnoseblock
LPDS: T     #LOOP_CNT_1;	//-> Schleifenzaehler
      LAR1  DID 38;	//Tippindex
      L     #ERROR_NO;	//Kanalnummer inkrementieren 
      INC   1;	//und in akt. Fach eintragen
      T     #ERROR_NO;
      L     DIB 48;	//Indexzaehler dekrementieren
      DEC   1;
      T     DIB 48;
      L     DID 38;	//Tippindex inkrementieren
      L     P#0.1;
      +D;
      T     DID 38;
      A     DIX [AR1,P#0.0];	//Wenn Bit fuer Kanal gesetzt
      JC    GFKL;	//-> Fehlerauswertung
      L     #LOOP_CNT_1;
      LOOP  LPDS;	//Wenn kein weiterer Fehler
      JU    BEND;	//-> Ende Diagnoseblock
//Kanalfehler wird gefunden im DS1
GFKL: LAR1  DID 52;	//Startadresse Diagnoseblock
      L     DIB [AR1,P#9.0];	//Anzahl der Diagnosebits pro Kanal
      SRW   3;	//: 8
      T     #TEMP_VAR_2;	//-> Anzahl Diagnosebytes sichern
      L     #ERROR_NO;	//x Kanalnummer
      *I;
      T     #TEMP_VAR_1;	//-> Offset des Kanals
      L     DIB [AR1,P#10.0];	//Anzahl der gleichart. Kanaele
      INC   7;	//+ 7
      L     8;	//: 8
      /I;	//-> Offset Kanalvektor
      L     #TEMP_VAR_1;
      +I;
      INC   11;	//+ Offset feste Daten
      SLD   3;
      +AR1;	//-> Adresse Kanalfehler-ID
      L     #TEMP_VAR_2;	//Anzahl Diagnosebytes pro Kanal
      JL    BYT0;	//ungueltiger Wert
